RoboDK station: kr30 cnc 072119 not table destroyer.rdk

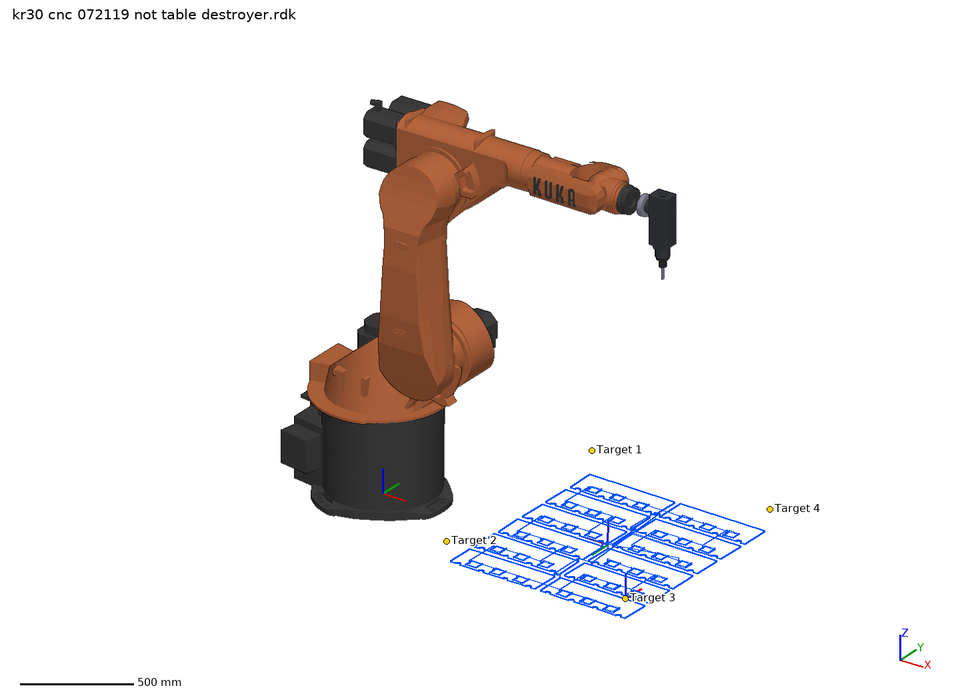
[picture v0: the station drawn from its stored meshes, robots at their saved joint values, targets as dots, program paths as lines]
Station kr30 cnc 072119 not table destroyer. Poses are relative to the parent item; angles as X-Y-Z fixed-axis rotations.
  - frame GIGASHEEN Base at (0, 0, 0) mm
    - robot GIGASHEEN (model KUKA KR 30 HA): 6 axes, payload 30 kg, reach 2033 mm, repeatability 0.05 mm, weight 665 kg
        modified DH rows (alpha deg, a mm, theta deg, d mm): 0, 0, 0, 815; -90, 350, 0, 0; 0, 850, -90, 0; -90, 145, 0, 820; 90, 0, 0, 0; -90, 0, 180, 170
        joint limits [-185, -135, -120, -350, -119, -350] to [185, 35, 158, 350, 119, 350]; home [0, -90, 90, 0, 0, 0]; saved at [0, -90, 90, 0, 0, 0]
      - tool 1/2" End Mill TCP, TCP at (337.71, -2.2, 160.57) mm, rotated rx 0 ry 90 rz 0 deg, size 415.8 x 102 x 153.6 mm
    - target Target 1 (joint target) at (982.46, 202.21, 406.25) mm, rotated rx -179.95 ry 0.15 rz -89.48 deg; joints [7.49, -59.642, 144.935, 97.969, -90.801, -4.608] of GIGASHEEN
    - target Target 2 (joint target) at (986.83, -921.64, 412.07) mm, rotated rx -179.94 ry 0.15 rz -89.48 deg; joints [51.766, -38.608, 94.384, 136.851, -116.554, -22.567] of GIGASHEEN
    - target Target 3 (joint target) at (1949.02, -919.97, 396.91) mm, rotated rx -179.94 ry 0.14 rz 179.61 deg; joints [29.5, -22.76, 62.288, 41.088, -47.759, -30.404] of GIGASHEEN
    - target Target 4 (joint target) at (1949.02, 190.94, 391.63) mm, rotated rx -179.94 ry 0.14 rz 179.61 deg; joints [-6.898, -35.989, 90.741, -8.88, -55.221, 5.167] of GIGASHEEN
  - machining project Machining Settings: C:/Users/liqui/OneDrive/Desktop/first half pipe jig.apt | rotZ(0) | rotX(0)*rotY(0) | rotZ(0)
  - program Prog2 (4 instructions, listed below)
  - frame Table at (1949.02, -919.97, 396.91) mm, rotated rx 0.87 ry 0.27 rz 90 deg
    - frame Frame 4 at (550, 480, -95) mm, rotated rx 0 ry 0 rz 90 deg
  - program Machining (1954 instructions, listed below)
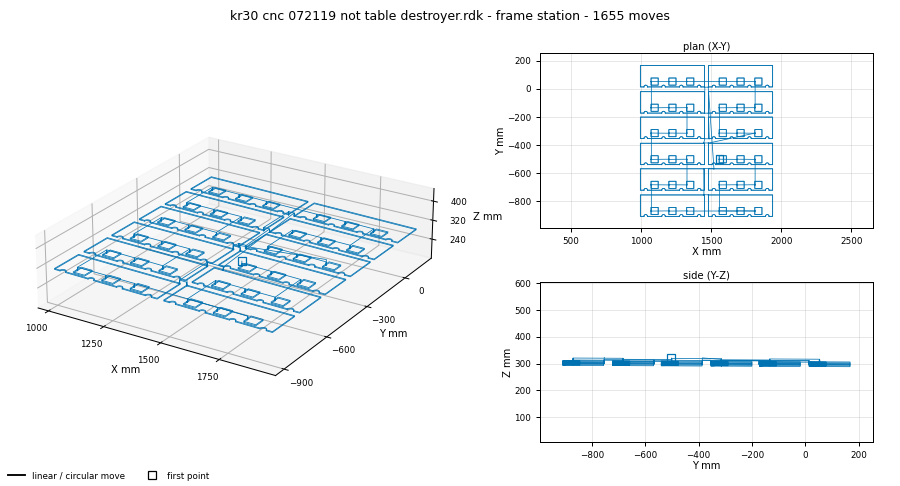
[picture p0: tool path of kr30 cnc 072119 not table destroyer.rdk in frame station, 1655 of 1659 moves have a stored position in this frame; points joined in program order, loops and branches not executed]

--- program Prog2 (robot GIGASHEEN) ---
  MoveJ (plywood back right safe) [its target is no longer in the station]
  MoveL (plywood back left safe) [its target is no longer in the station]
  MoveL (plywood front left safe) [its target is no longer in the station]
  MoveL (plywood front right safe) [its target is no longer in the station]

--- program Machining (robot GIGASHEEN) ---
  Smooth(0)
  Set Ref.: Frame 4
  Set Tool: 1/2" End Mill TCP
  Show 1/2" End Mill TCP
  Print: /'1001'
  Print: /''
  Print: /'2D Contour2'
  Set speed (500.0 mm/s)
  MoveJ 1 to (-92.16, 131.48, 15) mm, rotated rx -180 ry 0 rz 0 deg; joints [21.967, -44.262, 117.716, 22.916, -73.822, -6.095]
  MoveL 2 to (-92.16, 131.48, 15) mm, rotated rx -180 ry 0 rz 0 deg; joints [21.967, -44.262, 117.716, 22.916, -73.822, -6.095]
  MoveL 3 to (-92.16, 131.48, 15) mm, rotated rx -180 ry 0 rz 0 deg; joints [21.967, -44.262, 117.716, 22.916, -73.822, -6.095]
  Set speed (500.0 mm/s)
  MoveL 4 to (-92.16, 131.49, 6) mm, rotated rx -180 ry 0 rz 0 deg; joints [21.971, -43.695, 117.606, 22.87, -74.243, -5.911]
  Set speed (25.4 mm/s)
  MoveL 5 to (-92.16, 131.49, -3.54) mm, rotated rx -180 ry 0 rz 0 deg; joints [21.975, -43.092, 117.482, 22.822, -74.685, -5.719]
  MoveC 6 to (-91.98, 131.48, -3.99) mm, rotated rx -180 ry 0 rz 0 deg; joints [21.978, -43.069, 117.491, 22.822, -74.714, -5.707] to (-91.53, 131.48, -4.17) mm, rotated rx 180 ry 0 rz 0 deg; joints [21.986, -43.07, 117.523, 22.826, -74.743, -5.697]
  Set speed (50.8 mm/s)
  MoveL 7 to (-90.89, 131.48, -4.18) mm, rotated rx -180 ry 0 rz 0 deg; joints [21.996, -43.089, 117.572, 22.834, -74.772, -5.687]
  MoveC 8 to (-90.44, 131.3, -4.18) mm, rotated rx -180 ry 0 rz 0 deg; joints [21.996, -43.104, 117.612, 22.831, -74.796, -5.677] to (-90.26, 130.85, -4.17) mm, rotated rx 180 ry 0 rz 0 deg; joints [21.981, -43.115, 117.641, 22.813, -74.811, -5.666]
  MoveL 9 to (-90.26, 105.45, -4.18) mm, rotated rx -180 ry 0 rz 0 deg; joints [20.958, -43.388, 118.41, 21.71, -75.168, -5.214]
  MoveL 10 to (-141.06, 105.45, -4.18) mm, rotated rx -180 ry 0 rz 0 deg; joints [20.197, -41.862, 114.412, 21.181, -72.789, -5.949]
  MoveL 11 to (-141.06, 156.25, -4.18) mm, rotated rx -180 ry 0 rz 0 deg; joints [22.169, -41.28, 112.846, 23.353, -72.109, -6.929]
  MoveL 12 to (-90.26, 156.25, -4.17) mm, rotated rx -180 ry 0 rz 0 deg; joints [22.989, -42.824, 116.833, 23.909, -74.444, -6.139]
  MoveL 13 to (-90.26, 130.85, -4.17) mm, rotated rx 180 ry 0 rz 0 deg; joints [21.981, -43.115, 117.641, 22.813, -74.811, -5.666]
  MoveC 14 to (-90.44, 130.4, -4.18) mm, rotated rx -180 ry 0 rz 0 deg; joints [21.96, -43.114, 117.64, 22.792, -74.809, -5.661] to (-90.89, 130.21, -4.17) mm, rotated rx 180 ry 0 rz 0 deg; joints [21.945, -43.103, 117.611, 22.779, -74.79, -5.664]
  MoveL 15 to (-91.53, 130.21, -4.18) mm, rotated rx 180 ry 0 rz 0 deg; joints [21.935, -43.085, 117.562, 22.771, -74.761, -5.674]
  MoveC 16 to (-91.98, 130.21, -3.99) mm, rotated rx 180 ry 0 rz 0 deg; joints [21.928, -43.083, 117.53, 22.767, -74.732, -5.684] to (-92.16, 130.21, -3.54) mm, rotated rx -180 ry 0 rz 0 deg; joints [21.925, -43.106, 117.522, 22.767, -74.703, -5.696]
  Set speed (500.0 mm/s)
  MoveL 17 to (-92.16, 130.21, 5) mm, rotated rx 180 ry 0 rz 0 deg; joints [21.921, -43.646, 117.633, 22.809, -74.307, -5.867]
  MoveL 18 to (-92.16, 131.49, 5) mm, rotated rx -180 ry 0 rz 0 deg; joints [21.972, -43.632, 117.594, 22.864, -74.289, -5.891]
  Set speed (25.4 mm/s)
  MoveL 19 to (-92.16, 131.48, 1.82) mm, rotated rx 180 ry 0 rz 0 deg; joints [21.973, -43.431, 117.553, 22.848, -74.437, -5.827]
  MoveL 20 to (-92.16, 131.49, -7.72) mm, rotated rx -180 ry 0 rz 0 deg; joints [21.977, -42.828, 117.425, 22.802, -74.876, -5.636]
  MoveC 21 to (-91.98, 131.48, -8.16) mm, rotated rx -180 ry 0 rz 0 deg; joints [21.98, -42.804, 117.434, 22.802, -74.906, -5.624] to (-91.53, 131.48, -8.35) mm, rotated rx 180 ry 0 rz 0 deg; joints [21.988, -42.806, 117.466, 22.806, -74.935, -5.614]
  Set speed (50.8 mm/s)
  MoveL 22 to (-90.89, 131.48, -8.35) mm, rotated rx -180 ry 0 rz 0 deg; joints [21.998, -42.824, 117.515, 22.814, -74.964, -5.604]
  MoveC 23 to (-90.44, 131.3, -8.35) mm, rotated rx -180 ry 0 rz 0 deg; joints [21.998, -42.839, 117.555, 22.811, -74.988, -5.594] to (-90.26, 130.85, -8.35) mm, rotated rx 180 ry 0 rz 0 deg; joints [21.983, -42.85, 117.584, 22.794, -75.003, -5.583]
  MoveL 24 to (-90.26, 105.45, -8.35) mm, rotated rx -180 ry 0 rz 0 deg; joints [20.96, -43.121, 118.353, 21.691, -75.363, -5.134]
  MoveL 25 to (-141.06, 105.45, -8.35) mm, rotated rx -180 ry 0 rz 0 deg; joints [20.199, -41.606, 114.356, 21.161, -72.976, -5.874]
  MoveL 26 to (-141.06, 156.25, -8.35) mm, rotated rx -180 ry 0 rz 0 deg; joints [22.171, -41.027, 112.79, 23.33, -72.29, -6.848]
  MoveL 27 to (-90.26, 156.25, -8.35) mm, rotated rx -180 ry 0 rz 0 deg; joints [22.991, -42.562, 116.776, 23.888, -74.632, -6.053]
  MoveL 28 to (-90.26, 130.85, -8.35) mm, rotated rx 180 ry 0 rz 0 deg; joints [21.983, -42.85, 117.584, 22.794, -75.003, -5.583]
  MoveC 29 to (-90.44, 130.4, -8.35) mm, rotated rx 180 ry 0 rz 0 deg; joints [21.962, -42.849, 117.583, 22.772, -75.001, -5.578] to (-90.89, 130.21, -8.35) mm, rotated rx -180 ry 0 rz 0 deg; joints [21.947, -42.838, 117.554, 22.759, -74.983, -5.581]
  MoveL 30 to (-91.53, 130.21, -8.35) mm, rotated rx -180 ry 0 rz 0 deg; joints [21.937, -42.82, 117.505, 22.751, -74.953, -5.591]
  MoveC 31 to (-91.98, 130.21, -8.16) mm, rotated rx -180 ry 0 rz 0 deg; joints [21.93, -42.818, 117.473, 22.747, -74.924, -5.601] to (-92.16, 130.21, -7.72) mm, rotated rx 180 ry 0 rz 0 deg; joints [21.926, -42.842, 117.465, 22.747, -74.895, -5.613]
  Set speed (500.0 mm/s)
  MoveL 32 to (-92.16, 130.22, 6) mm, rotated rx -180 ry 0 rz 0 deg; joints [21.92, -43.71, 117.646, 22.814, -74.261, -5.888]
  MoveL 33 to (-219.16, 131.48, 6) mm, rotated rx 180 ry 0 rz 0 deg; joints [20.093, -39.587, 107.343, 21.691, -68.314, -7.771]
  Set speed (25.4 mm/s)
  MoveL 34 to (-219.16, 131.48, -3.54) mm, rotated rx -180 ry 0 rz 0 deg; joints [20.097, -39.042, 107.223, 21.633, -68.71, -7.604]
  MoveC 35 to (-218.98, 131.48, -3.99) mm, rotated rx 180 ry 0 rz 0 deg; joints [20.1, -39.022, 107.233, 21.632, -68.737, -7.593] to (-218.53, 131.48, -4.17) mm, rotated rx -180 ry 0 rz 0 deg; joints [20.106, -39.027, 107.269, 21.634, -68.767, -7.584]
  Set speed (50.8 mm/s)
  MoveL 36 to (-217.89, 131.48, -4.18) mm, rotated rx 180 ry 0 rz 0 deg; joints [20.115, -39.049, 107.322, 21.639, -68.797, -7.574]
  MoveC 37 to (-217.44, 131.3, -4.17) mm, rotated rx -180 ry 0 rz 0 deg; joints [20.114, -39.067, 107.366, 21.634, -68.821, -7.564] to (-217.26, 130.85, -4.17) mm, rotated rx -180 ry 0 rz 0 deg; joints [20.1, -39.079, 107.395, 21.617, -68.836, -7.551]
  MoveL 38 to (-217.26, 105.45, -4.18) mm, rotated rx -180 ry 0 rz 0 deg; joints [19.15, -39.375, 108.156, 20.544, -69.144, -7.025]
  MoveL 39 to (-268.06, 105.45, -4.18) mm, rotated rx 180 ry 0 rz 0 deg; joints [18.508, -37.578, 103.789, 20.221, -66.649, -7.743]
  MoveL 40 to (-268.06, 156.25, -4.18) mm, rotated rx 180 ry 0 rz 0 deg; joints [20.343, -36.949, 102.223, 22.351, -66.05, -8.881]
  MoveL 41 to (-217.26, 156.25, -4.17) mm, rotated rx -180 ry 0 rz 0 deg; joints [21.038, -38.765, 106.595, 22.685, -68.517, -8.097]
  MoveL 42 to (-217.26, 130.85, -4.17) mm, rotated rx -180 ry 0 rz 0 deg; joints [20.1, -39.079, 107.395, 21.617, -68.836, -7.551]
  MoveC 43 to (-217.44, 130.4, -4.17) mm, rotated rx -180 ry 0 rz 0 deg; joints [20.08, -39.078, 107.394, 21.596, -68.832, -7.545] to (-217.89, 130.21, -4.17) mm, rotated rx 180 ry 0 rz 0 deg; joints [20.067, -39.064, 107.361, 21.585, -68.813, -7.547]
  MoveL 44 to (-218.53, 130.21, -4.18) mm, rotated rx -180 ry 0 rz 0 deg; joints [20.059, -39.042, 107.308, 21.581, -68.782, -7.557]
  MoveC 45 to (-218.98, 130.21, -3.99) mm, rotated rx -180 ry 0 rz 0 deg; joints [20.053, -39.038, 107.272, 21.578, -68.753, -7.567] to (-219.16, 130.21, -3.54) mm, rotated rx 180 ry 0 rz 0 deg; joints [20.05, -39.057, 107.262, 21.58, -68.725, -7.577]
  Set speed (500.0 mm/s)
  MoveL 46 to (-219.16, 130.21, 5) mm, rotated rx 180 ry 0 rz 0 deg; joints [20.047, -39.545, 107.37, 21.631, -68.371, -7.727]
  MoveL 47 to (-219.16, 131.48, 5) mm, rotated rx 180 ry 0 rz 0 deg; joints [20.094, -39.53, 107.331, 21.685, -68.355, -7.754]
  Set speed (25.4 mm/s)
  MoveL 48 to (-219.16, 131.48, 1.83) mm, rotated rx -180 ry 0 rz 0 deg; joints [20.095, -39.348, 107.291, 21.666, -68.488, -7.698]
  MoveL 49 to (-219.16, 131.48, -7.72) mm, rotated rx 180 ry 0 rz 0 deg; joints [20.099, -38.802, 107.169, 21.609, -68.882, -7.532]
  MoveC 50 to (-218.98, 131.49, -8.16) mm, rotated rx -180 ry 0 rz 0 deg; joints [20.101, -38.783, 107.179, 21.607, -68.909, -7.521] to (-218.53, 131.48, -8.35) mm, rotated rx -180 ry 0 rz 0 deg; joints [20.108, -38.788, 107.214, 21.609, -68.939, -7.511]
  Set speed (50.8 mm/s)
  MoveL 51 to (-217.89, 131.48, -8.35) mm, rotated rx -180 ry 0 rz 0 deg; joints [20.116, -38.81, 107.268, 21.614, -68.969, -7.502]
  MoveC 52 to (-217.44, 131.3, -8.35) mm, rotated rx 180 ry 0 rz 0 deg; joints [20.115, -38.827, 107.311, 21.61, -68.993, -7.491] to (-217.26, 130.85, -8.35) mm, rotated rx 180 ry 0 rz 0 deg; joints [20.101, -38.839, 107.341, 21.592, -69.008, -7.479]
  MoveL 53 to (-217.26, 105.45, -8.35) mm, rotated rx -180 ry 0 rz 0 deg; joints [19.151, -39.133, 108.101, 20.521, -69.319, -6.956]
  MoveL 54 to (-268.06, 105.45, -8.35) mm, rotated rx -180 ry 0 rz 0 deg; joints [18.509, -37.346, 103.734, 20.196, -66.816, -7.677]
  MoveL 55 to (-268.06, 156.25, -8.35) mm, rotated rx 180 ry 0 rz 0 deg; joints [20.345, -36.72, 102.169, 22.323, -66.212, -8.809]
  MoveL 56 to (-217.26, 156.25, -8.35) mm, rotated rx -180 ry 0 rz 0 deg; joints [21.04, -38.527, 106.541, 22.659, -68.687, -8.021]
  MoveL 57 to (-217.26, 130.85, -8.35) mm, rotated rx 180 ry 0 rz 0 deg; joints [20.101, -38.839, 107.341, 21.592, -69.008, -7.479]
  MoveC 58 to (-217.44, 130.4, -8.35) mm, rotated rx 180 ry 0 rz 0 deg; joints [20.082, -38.838, 107.339, 21.572, -69.005, -7.472] to (-217.89, 130.22, -8.35) mm, rotated rx -180 ry 0 rz 0 deg; joints [20.069, -38.825, 107.307, 21.561, -68.985, -7.475]
  MoveL 59 to (-218.53, 130.22, -8.35) mm, rotated rx -180 ry 0 rz 0 deg; joints [20.06, -38.803, 107.253, 21.556, -68.954, -7.485]
  MoveC 60 to (-218.98, 130.21, -8.16) mm, rotated rx -180 ry 0 rz 0 deg; joints [20.054, -38.798, 107.218, 21.554, -68.925, -7.494] to (-219.16, 130.22, -7.72) mm, rotated rx -180 ry 0 rz 0 deg; joints [20.051, -38.818, 107.208, 21.555, -68.898, -7.505]
  Set speed (500.0 mm/s)
  MoveL 61 to (-219.16, 130.21, 6) mm, rotated rx -180 ry 0 rz 0 deg; joints [20.046, -39.602, 107.382, 21.638, -68.329, -7.744]
  MoveL 62 to (-346.16, 131.48, 6) mm, rotated rx -180 ry 0 rz 0 deg; joints [18.501, -34.783, 96.043, 21.052, -62.014, -9.675]
  Set speed (25.4 mm/s)
  MoveL 63 to (-346.16, 131.48, -3.54) mm, rotated rx -180 ry 0 rz 0 deg; joints [18.504, -34.284, 95.924, 20.984, -62.369, -9.523]
  MoveC 64 to (-345.98, 131.48, -3.99) mm, rotated rx -180 ry 0 rz 0 deg; joints [18.507, -34.269, 95.936, 20.982, -62.395, -9.513] to (-345.53, 131.48, -4.17) mm, rotated rx 180 ry 0 rz 0 deg; joints [18.512, -34.277, 95.975, 20.982, -62.426, -9.503]
  Set speed (50.8 mm/s)
  MoveL 65 to (-344.89, 131.48, -4.18) mm, rotated rx -180 ry 0 rz 0 deg; joints [18.519, -34.303, 96.035, 20.983, -62.458, -9.493]
  MoveC 66 to (-344.44, 131.3, -4.17) mm, rotated rx -180 ry 0 rz 0 deg; joints [18.518, -34.323, 96.083, 20.977, -62.484, -9.481] to (-344.26, 130.85, -4.17) mm, rotated rx -180 ry 0 rz 0 deg; joints [18.504, -34.337, 96.115, 20.959, -62.498, -9.467]
  MoveL 67 to (-344.26, 105.45, -4.18) mm, rotated rx -180 ry 0 rz 0 deg; joints [17.62, -34.658, 96.888, 19.894, -62.777, -8.851]
  MoveL 68 to (-395.06, 105.45, -4.17) mm, rotated rx -180 ry 0 rz 0 deg; joints [17.072, -32.543, 92.01, 19.79, -60.088, -9.633]
  MoveL 69 to (-395.06, 156.25, -4.18) mm, rotated rx -180 ry 0 rz 0 deg; joints [18.786, -31.855, 90.392, 21.931, -59.533, -10.971]
  MoveL 70 to (-344.26, 156.25, -4.18) mm, rotated rx -180 ry 0 rz 0 deg; joints [19.38, -33.996, 95.299, 22.023, -62.209, -10.102]
  MoveL 71 to (-344.26, 130.85, -4.17) mm, rotated rx -180 ry 0 rz 0 deg; joints [18.504, -34.337, 96.115, 20.959, -62.498, -9.467]
  MoveC 72 to (-344.44, 130.4, -4.18) mm, rotated rx -180 ry 0 rz 0 deg; joints [18.487, -34.335, 96.111, 20.939, -62.494, -9.459] to (-344.89, 130.21, -4.18) mm, rotated rx 180 ry 0 rz 0 deg; joints [18.475, -34.319, 96.075, 20.93, -62.473, -9.462]
  MoveL 73 to (-345.53, 130.21, -4.18) mm, rotated rx -180 ry 0 rz 0 deg; joints [18.468, -34.294, 96.015, 20.928, -62.44, -9.472]
  MoveC 74 to (-345.98, 130.22, -3.99) mm, rotated rx -180 ry 0 rz 0 deg; joints [18.463, -34.285, 95.975, 20.928, -62.41, -9.482] to (-346.16, 130.21, -3.54) mm, rotated rx -180 ry 0 rz 0 deg; joints [18.46, -34.301, 95.964, 20.931, -62.383, -9.492]
  Set speed (500.0 mm/s)
  MoveL 75 to (-346.16, 130.21, 5) mm, rotated rx -180 ry 0 rz 0 deg; joints [18.457, -34.748, 96.07, 20.992, -62.065, -9.628]
  MoveL 76 to (-346.16, 131.48, 5) mm, rotated rx -180 ry 0 rz 0 deg; joints [18.501, -34.731, 96.031, 21.045, -62.051, -9.659]
  Set speed (25.4 mm/s)
  MoveL 77 to (-346.16, 131.48, 1.82) mm, rotated rx -180 ry 0 rz 0 deg; joints [18.502, -34.565, 95.992, 21.022, -62.17, -9.608]
  MoveL 78 to (-346.16, 131.48, -7.71) mm, rotated rx 180 ry 0 rz 0 deg; joints [18.506, -34.065, 95.87, 20.955, -62.523, -9.457]
  MoveC 79 to (-345.98, 131.48, -8.16) mm, rotated rx -180 ry 0 rz 0 deg; joints [18.508, -34.049, 95.881, 20.952, -62.549, -9.447] to (-345.53, 131.48, -8.35) mm, rotated rx -180 ry 0 rz 0 deg; joints [18.513, -34.058, 95.921, 20.952, -62.58, -9.437]
  Set speed (50.8 mm/s)
  MoveL 80 to (-344.89, 131.48, -8.35) mm, rotated rx -180 ry 0 rz 0 deg; joints [18.521, -34.083, 95.981, 20.954, -62.613, -9.427]
  MoveC 81 to (-344.44, 131.3, -8.35) mm, rotated rx -180 ry 0 rz 0 deg; joints [18.519, -34.104, 96.029, 20.948, -62.638, -9.415] to (-344.26, 130.85, -8.35) mm, rotated rx 180 ry 0 rz 0 deg; joints [18.506, -34.117, 96.06, 20.93, -62.653, -9.401]
  MoveL 82 to (-344.26, 105.45, -8.35) mm, rotated rx -180 ry 0 rz 0 deg; joints [17.621, -34.437, 96.833, 19.867, -62.934, -8.788]
  MoveL 83 to (-395.06, 105.45, -8.35) mm, rotated rx -180 ry 0 rz 0 deg; joints [17.073, -32.329, 91.955, 19.76, -60.238, -9.572]
  MoveL 84 to (-395.06, 156.25, -8.35) mm, rotated rx -180 ry 0 rz 0 deg; joints [18.787, -31.643, 90.337, 21.899, -59.678, -10.904]
  MoveL 85 to (-344.26, 156.25, -8.35) mm, rotated rx -180 ry 0 rz 0 deg; joints [19.382, -33.778, 95.244, 21.993, -62.361, -10.034]
  MoveL 86 to (-344.26, 130.85, -8.35) mm, rotated rx 180 ry 0 rz 0 deg; joints [18.506, -34.117, 96.06, 20.93, -62.653, -9.401]
  MoveC 87 to (-344.44, 130.4, -8.35) mm, rotated rx -180 ry 0 rz 0 deg; joints [18.488, -34.115, 96.057, 20.91, -62.648, -9.393] to (-344.89, 130.21, -8.35) mm, rotated rx -180 ry 0 rz 0 deg; joints [18.477, -34.1, 96.02, 20.901, -62.627, -9.396]
  MoveL 88 to (-345.53, 130.21, -8.35) mm, rotated rx -180 ry 0 rz 0 deg; joints [18.469, -34.074, 95.961, 20.899, -62.594, -9.406]
  MoveC 89 to (-345.98, 130.21, -8.16) mm, rotated rx -180 ry 0 rz 0 deg; joints [18.464, -34.066, 95.921, 20.899, -62.564, -9.416] to (-346.16, 130.21, -7.72) mm, rotated rx 180 ry 0 rz 0 deg; joints [18.462, -34.082, 95.909, 20.902, -62.538, -9.426]
  Set speed (500.0 mm/s)
  MoveL 90 to (-346.16, 130.21, 6) mm, rotated rx 180 ry 0 rz 0 deg; joints [18.457, -34.8, 96.082, 20.999, -62.028, -9.644]
  MoveL 91 to (-346.16, 313.35, 6) mm, rotated rx -180 ry 0 rz 0 deg; joints [24.551, -31.864, 89.216, 28.735, -59.772, -14.762]
  Set speed (25.4 mm/s)
  MoveL 92 to (-346.16, 313.35, -3.54) mm, rotated rx -180 ry 0 rz 0 deg; joints [24.555, -31.387, 89.095, 28.64, -60.086, -14.565]
  MoveC 93 to (-345.98, 313.35, -3.99) mm, rotated rx -180 ry 0 rz 0 deg; joints [24.557, -31.372, 89.107, 28.636, -60.11, -14.552] to (-345.53, 313.35, -4.17) mm, rotated rx 180 ry 0 rz 0 deg; joints [24.564, -31.382, 89.148, 28.634, -60.139, -14.539]
  Set speed (50.8 mm/s)
  MoveL 94 to (-344.89, 313.35, -4.18) mm, rotated rx 180 ry 0 rz 0 deg; joints [24.573, -31.409, 89.21, 28.635, -60.171, -14.525]
  MoveC 95 to (-344.44, 313.17, -4.18) mm, rotated rx 180 ry 0 rz 0 deg; joints [24.574, -31.432, 89.261, 28.628, -60.197, -14.509] to (-344.26, 312.72, -4.18) mm, rotated rx 180 ry 0 rz 0 deg; joints [24.562, -31.448, 89.299, 28.609, -60.213, -14.491]
  MoveL 96 to (-344.26, 287.32, -4.18) mm, rotated rx -180 ry 0 rz 0 deg; joints [23.747, -31.917, 90.391, 27.535, -60.56, -13.718]
  MoveL 97 to (-395.06, 287.32, -4.17) mm, rotated rx -180 ry 0 rz 0 deg; joints [23.046, -29.688, 85.37, 27.512, -57.909, -14.825]
  MoveL 98 to (-395.06, 338.12, -4.18) mm, rotated rx -180 ry 0 rz 0 deg; joints [24.63, -28.683, 83.075, 29.71, -57.21, -16.501]
  MoveL 99 to (-344.26, 338.12, -4.18) mm, rotated rx -180 ry 0 rz 0 deg; joints [25.367, -30.956, 88.159, 29.688, -59.857, -15.291]
  MoveL 100 to (-344.26, 312.72, -4.17) mm, rotated rx -180 ry 0 rz 0 deg; joints [24.562, -31.448, 89.299, 28.609, -60.213, -14.491]
  MoveC 101 to (-344.44, 312.27, -4.18) mm, rotated rx -180 ry 0 rz 0 deg; joints [24.545, -31.449, 89.301, 28.59, -60.209, -14.481] to (-344.89, 312.08, -4.18) mm, rotated rx -180 ry 0 rz 0 deg; joints [24.533, -31.433, 89.265, 28.581, -60.189, -14.485]
  MoveL 102 to (-345.53, 312.08, -4.17) mm, rotated rx -180 ry 0 rz 0 deg; joints [24.524, -31.406, 89.204, 28.581, -60.157, -14.499]
  MoveC 103 to (-345.98, 312.08, -3.99) mm, rotated rx -180 ry 0 rz 0 deg; joints [24.517, -31.396, 89.163, 28.582, -60.128, -14.513] to (-346.16, 312.08, -3.54) mm, rotated rx -180 ry 0 rz 0 deg; joints [24.514, -31.411, 89.151, 28.586, -60.103, -14.526]
  Set speed (500.0 mm/s)
  MoveL 104 to (-346.16, 312.08, 5) mm, rotated rx -180 ry 0 rz 0 deg; joints [24.511, -31.838, 89.259, 28.671, -59.822, -14.701]
  MoveL 105 to (-346.16, 313.35, 5) mm, rotated rx 180 ry 0 rz 0 deg; joints [24.551, -31.814, 89.203, 28.725, -59.805, -14.741]
  Set speed (25.4 mm/s)
  MoveL 106 to (-346.16, 313.35, 1.82) mm, rotated rx 180 ry 0 rz 0 deg; joints [24.553, -31.655, 89.164, 28.693, -59.91, -14.675]
  MoveL 107 to (-346.16, 313.35, -7.72) mm, rotated rx 180 ry 0 rz 0 deg; joints [24.556, -31.177, 89.04, 28.599, -60.222, -14.481]
  MoveC 108 to (-345.98, 313.35, -8.16) mm, rotated rx -180 ry 0 rz 0 deg; joints [24.559, -31.162, 89.052, 28.595, -60.246, -14.468] to (-345.53, 313.35, -8.35) mm, rotated rx -180 ry 0 rz 0 deg; joints [24.566, -31.172, 89.093, 28.594, -60.275, -14.454]
  Set speed (50.8 mm/s)
  MoveL 109 to (-344.89, 313.35, -8.35) mm, rotated rx -180 ry 0 rz 0 deg; joints [24.575, -31.199, 89.154, 28.595, -60.308, -14.44]
  MoveC 110 to (-344.44, 313.17, -8.35) mm, rotated rx 180 ry 0 rz 0 deg; joints [24.575, -31.221, 89.206, 28.587, -60.333, -14.425] to (-344.26, 312.72, -8.35) mm, rotated rx 180 ry 0 rz 0 deg; joints [24.564, -31.238, 89.244, 28.569, -60.349, -14.407]
  MoveL 111 to (-344.26, 287.32, -8.35) mm, rotated rx -180 ry 0 rz 0 deg; joints [23.749, -31.705, 90.335, 27.496, -60.699, -13.636]
  MoveL 112 to (-395.06, 287.32, -8.35) mm, rotated rx -180 ry 0 rz 0 deg; joints [23.047, -29.482, 85.314, 27.471, -58.042, -14.744]
  MoveL 113 to (-395.06, 338.12, -8.35) mm, rotated rx -180 ry 0 rz 0 deg; joints [24.631, -28.479, 83.018, 29.665, -57.338, -16.416]
  MoveL 114 to (-344.26, 338.12, -8.35) mm, rotated rx 180 ry 0 rz 0 deg; joints [25.369, -30.747, 88.104, 29.645, -59.991, -15.204]
  MoveL 115 to (-344.26, 312.72, -8.35) mm, rotated rx 180 ry 0 rz 0 deg; joints [24.564, -31.238, 89.244, 28.569, -60.349, -14.407]
  MoveC 116 to (-344.44, 312.27, -8.35) mm, rotated rx -180 ry 0 rz 0 deg; joints [24.547, -31.238, 89.245, 28.549, -60.346, -14.397] to (-344.89, 312.08, -8.35) mm, rotated rx -180 ry 0 rz 0 deg; joints [24.534, -31.223, 89.21, 28.541, -60.326, -14.401]
  MoveL 117 to (-345.53, 312.08, -8.35) mm, rotated rx -180 ry 0 rz 0 deg; joints [24.525, -31.196, 89.149, 28.54, -60.293, -14.415]
  MoveC 118 to (-345.98, 312.08, -8.16) mm, rotated rx -180 ry 0 rz 0 deg; joints [24.518, -31.186, 89.108, 28.541, -60.264, -14.428] to (-346.16, 312.08, -7.72) mm, rotated rx 180 ry 0 rz 0 deg; joints [24.516, -31.201, 89.096, 28.545, -60.24, -14.441]
  Set speed (500.0 mm/s)
  MoveL 119 to (-346.16, 312.08, 6) mm, rotated rx 180 ry 0 rz 0 deg; joints [24.511, -31.888, 89.271, 28.681, -59.789, -14.722]
  MoveL 120 to (-219.16, 313.35, 6) mm, rotated rx 180 ry 0 rz 0 deg; joints [26.538, -36.893, 100.706, 29.297, -65.896, -12.2]
  Set speed (25.4 mm/s)
  MoveL 121 to (-219.16, 313.35, -3.54) mm, rotated rx 180 ry 0 rz 0 deg; joints [26.542, -36.378, 100.588, 29.215, -66.244, -11.989]
  MoveC 122 to (-218.98, 313.36, -3.99) mm, rotated rx -180 ry 0 rz 0 deg; joints [26.545, -36.36, 100.598, 29.213, -66.268, -11.976] to (-218.53, 313.36, -4.17) mm, rotated rx -180 ry 0 rz 0 deg; joints [26.553, -36.366, 100.634, 29.214, -66.296, -11.963]
  Set speed (50.8 mm/s)
  MoveL 123 to (-217.89, 313.36, -4.17) mm, rotated rx -180 ry 0 rz 0 deg; joints [26.563, -36.389, 100.688, 29.219, -66.325, -11.951]
  MoveC 124 to (-217.44, 313.17, -4.17) mm, rotated rx -180 ry 0 rz 0 deg; joints [26.565, -36.408, 100.734, 29.215, -66.349, -11.937] to (-217.26, 312.72, -4.17) mm, rotated rx 180 ry 0 rz 0 deg; joints [26.553, -36.423, 100.769, 29.198, -66.364, -11.922]
  MoveL 125 to (-217.26, 287.32, -4.18) mm, rotated rx -180 ry 0 rz 0 deg; joints [25.689, -36.853, 101.821, 28.148, -66.733, -11.243]
  MoveL 126 to (-268.06, 287.32, -4.18) mm, rotated rx 180 ry 0 rz 0 deg; joints [24.878, -34.977, 97.416, 27.815, -64.331, -12.197]
  MoveL 127 to (-268.06, 338.12, -4.18) mm, rotated rx 180 ry 0 rz 0 deg; joints [26.553, -34.068, 95.246, 29.928, -63.609, -13.647]
  MoveL 128 to (-217.26, 338.12, -4.18) mm, rotated rx 180 ry 0 rz 0 deg; joints [27.403, -35.973, 99.674, 30.246, -65.989, -12.625]
  MoveL 129 to (-217.26, 312.72, -4.17) mm, rotated rx 180 ry 0 rz 0 deg; joints [26.553, -36.423, 100.769, 29.198, -66.364, -11.922]
  MoveC 130 to (-217.44, 312.27, -4.17) mm, rotated rx -180 ry 0 rz 0 deg; joints [26.534, -36.424, 100.772, 29.178, -66.362, -11.913] to (-217.89, 312.08, -4.18) mm, rotated rx 180 ry 0 rz 0 deg; joints [26.52, -36.411, 100.742, 29.167, -66.344, -11.917]
  MoveL 131 to (-218.53, 312.08, -4.17) mm, rotated rx -180 ry 0 rz 0 deg; joints [26.51, -36.388, 100.688, 29.162, -66.315, -11.929]
  MoveC 132 to (-218.98, 312.08, -3.99) mm, rotated rx -180 ry 0 rz 0 deg; joints [26.502, -36.382, 100.652, 29.16, -66.287, -11.941] to (-219.16, 312.08, -3.54) mm, rotated rx -180 ry 0 rz 0 deg; joints [26.499, -36.4, 100.642, 29.163, -66.262, -11.955]
  Set speed (500.0 mm/s)
  MoveL 133 to (-219.16, 312.08, 5) mm, rotated rx -180 ry 0 rz 0 deg; joints [26.495, -36.862, 100.748, 29.236, -65.951, -12.143]
  MoveL 134 to (-219.16, 313.35, 5) mm, rotated rx -180 ry 0 rz 0 deg; joints [26.538, -36.839, 100.694, 29.288, -65.932, -12.178]
  Set speed (25.4 mm/s)
  MoveL 135 to (-219.16, 313.35, 1.83) mm, rotated rx -180 ry 0 rz 0 deg; joints [26.539, -36.668, 100.655, 29.261, -66.048, -12.107]
  MoveL 136 to (-219.16, 313.35, -7.71) mm, rotated rx -180 ry 0 rz 0 deg; joints [26.543, -36.151, 100.534, 29.18, -66.395, -11.898]
  MoveC 137 to (-218.98, 313.35, -8.16) mm, rotated rx -180 ry 0 rz 0 deg; joints [26.547, -36.133, 100.544, 29.178, -66.419, -11.885] to (-218.53, 313.35, -8.35) mm, rotated rx -180 ry 0 rz 0 deg; joints [26.554, -36.139, 100.58, 29.179, -66.447, -11.872]
  Set speed (50.8 mm/s)
  MoveL 138 to (-217.89, 313.35, -8.35) mm, rotated rx -180 ry 0 rz 0 deg; joints [26.565, -36.162, 100.634, 29.184, -66.476, -11.86]
  MoveC 139 to (-217.44, 313.17, -8.35) mm, rotated rx -180 ry 0 rz 0 deg; joints [26.566, -36.181, 100.68, 29.18, -66.5, -11.846] to (-217.26, 312.72, -8.35) mm, rotated rx -180 ry 0 rz 0 deg; joints [26.554, -36.196, 100.714, 29.163, -66.515, -11.83]
  MoveL 140 to (-217.26, 287.32, -8.35) mm, rotated rx -180 ry 0 rz 0 deg; joints [25.691, -36.624, 101.767, 28.114, -66.887, -11.154]
  MoveL 141 to (-268.06, 287.32, -8.35) mm, rotated rx -180 ry 0 rz 0 deg; joints [24.88, -34.755, 97.362, 27.78, -64.479, -12.112]
  MoveL 142 to (-268.06, 338.12, -8.35) mm, rotated rx 180 ry 0 rz 0 deg; joints [26.555, -33.85, 95.192, 29.889, -63.751, -13.556]
  MoveL 143 to (-217.26, 338.12, -8.35) mm, rotated rx 180 ry 0 rz 0 deg; joints [27.404, -35.748, 99.62, 30.21, -66.137, -12.531]
  MoveL 144 to (-217.26, 312.72, -8.35) mm, rotated rx -180 ry 0 rz 0 deg; joints [26.554, -36.196, 100.714, 29.163, -66.515, -11.83]
  MoveC 145 to (-217.44, 312.27, -8.35) mm, rotated rx 180 ry 0 rz 0 deg; joints [26.536, -36.197, 100.718, 29.143, -66.513, -11.822] to (-217.89, 312.09, -8.35) mm, rotated rx -180 ry 0 rz 0 deg; joints [26.522, -36.184, 100.687, 29.132, -66.495, -11.825]
  MoveL 146 to (-218.53, 312.08, -8.35) mm, rotated rx 180 ry 0 rz 0 deg; joints [26.511, -36.161, 100.633, 29.127, -66.466, -11.838]
  MoveC 147 to (-218.98, 312.08, -8.16) mm, rotated rx -180 ry 0 rz 0 deg; joints [26.504, -36.155, 100.598, 29.125, -66.438, -11.85] to (-219.16, 312.08, -7.72) mm, rotated rx 180 ry 0 rz 0 deg; joints [26.501, -36.173, 100.588, 29.128, -66.413, -11.864]
  Set speed (500.0 mm/s)
  MoveL 148 to (-219.16, 312.08, 6) mm, rotated rx -180 ry 0 rz 0 deg; joints [26.495, -36.916, 100.76, 29.244, -65.914, -12.165]
  MoveL 149 to (-92.16, 313.35, 6) mm, rotated rx -180 ry 0 rz 0 deg; joints [28.844, -41.18, 110.953, 30.568, -71.515, -9.856]
  Set speed (25.4 mm/s)
  MoveL 150 to (-92.16, 313.35, -3.54) mm, rotated rx -180 ry 0 rz 0 deg; joints [28.849, -40.617, 110.833, 30.498, -71.897, -9.62]
  MoveC 151 to (-91.98, 313.36, -3.99) mm, rotated rx 180 ry 0 rz 0 deg; joints [28.853, -40.596, 110.842, 30.497, -71.923, -9.605] to (-91.53, 313.36, -4.17) mm, rotated rx -180 ry 0 rz 0 deg; joints [28.862, -40.599, 110.874, 30.501, -71.95, -9.593]
  Set speed (50.8 mm/s)
  MoveL 152 to (-90.89, 313.36, -4.18) mm, rotated rx -180 ry 0 rz 0 deg; joints [28.874, -40.618, 110.922, 30.509, -71.977, -9.581]
  MoveC 153 to (-90.44, 313.17, -4.18) mm, rotated rx 180 ry 0 rz 0 deg; joints [28.876, -40.635, 110.964, 30.507, -71.999, -9.568] to (-90.26, 312.72, -4.17) mm, rotated rx 180 ry 0 rz 0 deg; joints [28.864, -40.648, 110.997, 30.491, -72.015, -9.553]
  MoveL 154 to (-90.26, 287.32, -4.18) mm, rotated rx -180 ry 0 rz 0 deg; joints [27.95, -41.048, 112.045, 29.442, -72.424, -8.939]
  MoveL 155 to (-141.06, 287.32, -4.17) mm, rotated rx -180 ry 0 rz 0 deg; joints [27.003, -39.45, 108.078, 28.846, -70.196, -9.855]
  MoveL 156 to (-141.06, 338.12, -4.18) mm, rotated rx 180 ry 0 rz 0 deg; joints [28.775, -38.608, 105.945, 30.937, -69.409, -11.154]
  MoveL 157 to (-90.26, 338.12, -4.17) mm, rotated rx -180 ry 0 rz 0 deg; joints [29.762, -40.229, 109.911, 31.535, -71.6, -10.192]
  MoveL 158 to (-90.26, 312.72, -4.17) mm, rotated rx 180 ry 0 rz 0 deg; joints [28.864, -40.648, 110.997, 30.491, -72.015, -9.553]
  MoveC 159 to (-90.44, 312.27, -4.17) mm, rotated rx -180 ry 0 rz 0 deg; joints [28.844, -40.65, 111.002, 30.47, -72.014, -9.546] to (-90.89, 312.08, -4.18) mm, rotated rx 180 ry 0 rz 0 deg; joints [28.829, -40.639, 110.976, 30.457, -71.998, -9.549]
  MoveL 160 to (-91.53, 312.08, -4.18) mm, rotated rx -180 ry 0 rz 0 deg; joints [28.816, -40.619, 110.927, 30.449, -71.97, -9.561]
  MoveC 161 to (-91.98, 312.08, -3.99) mm, rotated rx 180 ry 0 rz 0 deg; joints [28.808, -40.616, 110.895, 30.445, -71.944, -9.574] to (-92.16, 312.08, -3.54) mm, rotated rx -180 ry 0 rz 0 deg; joints [28.804, -40.637, 110.886, 30.445, -71.918, -9.588]
  Set speed (500.0 mm/s)
  MoveL 162 to (-92.16, 312.08, 5) mm, rotated rx 180 ry 0 rz 0 deg; joints [28.8, -41.142, 110.994, 30.508, -71.575, -9.799]
  MoveL 163 to (-92.16, 313.35, 5) mm, rotated rx -180 ry 0 rz 0 deg; joints [28.845, -41.121, 110.941, 30.56, -71.555, -9.831]
  Set speed (25.4 mm/s)
  MoveL 164 to (-92.16, 313.36, 1.82) mm, rotated rx -180 ry 0 rz 0 deg; joints [28.846, -40.934, 110.902, 30.537, -71.683, -9.752]
  MoveL 165 to (-92.16, 313.35, -7.72) mm, rotated rx -180 ry 0 rz 0 deg; joints [28.851, -40.37, 110.778, 30.468, -72.063, -9.518]
  MoveC 166 to (-91.98, 313.35, -8.16) mm, rotated rx -180 ry 0 rz 0 deg; joints [28.855, -40.349, 110.786, 30.467, -72.089, -9.503] to (-91.53, 313.35, -8.35) mm, rotated rx 180 ry 0 rz 0 deg; joints [28.864, -40.351, 110.818, 30.472, -72.116, -9.491]
  Set speed (50.8 mm/s)
  MoveL 167 to (-90.89, 313.35, -8.35) mm, rotated rx -180 ry 0 rz 0 deg; joints [28.876, -40.371, 110.867, 30.48, -72.143, -9.479]
  MoveC 168 to (-90.44, 313.17, -8.35) mm, rotated rx -180 ry 0 rz 0 deg; joints [28.878, -40.387, 110.909, 30.478, -72.166, -9.466] to (-90.26, 312.72, -8.35) mm, rotated rx -180 ry 0 rz 0 deg; joints [28.866, -40.4, 110.942, 30.462, -72.181, -9.451]
  MoveL 169 to (-90.26, 287.32, -8.35) mm, rotated rx -180 ry 0 rz 0 deg; joints [27.952, -40.798, 111.99, 29.413, -72.594, -8.839]
  MoveL 170 to (-141.06, 287.32, -8.35) mm, rotated rx -180 ry 0 rz 0 deg; joints [27.005, -39.209, 108.023, 28.816, -70.36, -9.76]
  MoveL 171 to (-141.06, 338.12, -8.35) mm, rotated rx -180 ry 0 rz 0 deg; joints [28.777, -38.371, 105.891, 30.904, -69.565, -11.054]
  MoveL 172 to (-90.26, 338.12, -8.35) mm, rotated rx -180 ry 0 rz 0 deg; joints [29.764, -39.984, 109.856, 31.504, -71.763, -10.088]
  MoveL 173 to (-90.26, 312.72, -8.35) mm, rotated rx -180 ry 0 rz 0 deg; joints [28.866, -40.4, 110.942, 30.462, -72.181, -9.451]
  MoveC 174 to (-90.44, 312.27, -8.35) mm, rotated rx -180 ry 0 rz 0 deg; joints [28.846, -40.402, 110.947, 30.441, -72.18, -9.444] to (-90.89, 312.08, -8.35) mm, rotated rx 180 ry 0 rz 0 deg; joints [28.831, -40.391, 110.92, 30.428, -72.164, -9.448]
  MoveL 175 to (-91.53, 312.08, -8.35) mm, rotated rx -180 ry 0 rz 0 deg; joints [28.818, -40.372, 110.872, 30.419, -72.137, -9.459]
  MoveC 176 to (-91.98, 312.08, -8.16) mm, rotated rx -180 ry 0 rz 0 deg; joints [28.809, -40.369, 110.84, 30.415, -72.11, -9.472] to (-92.16, 312.09, -7.72) mm, rotated rx -180 ry 0 rz 0 deg; joints [28.806, -40.39, 110.832, 30.416, -72.084, -9.487]
  Set speed (500.0 mm/s)
  MoveL 177 to (-92.16, 312.08, 6) mm, rotated rx -180 ry 0 rz 0 deg; joints [28.799, -41.201, 111.007, 30.515, -71.535, -9.824]
  MoveL 178 to (-92.16, 499.69, 6) mm, rotated rx 180 ry 0 rz 0 deg; joints [35.058, -37.589, 102.036, 38.119, -68.484, -15.172]
  Set speed (25.4 mm/s)
  MoveL 179 to (-92.16, 499.69, -3.54) mm, rotated rx -180 ry 0 rz 0 deg; joints [35.062, -37.068, 101.919, 38.026, -68.803, -14.906]
  MoveC 180 to (-91.98, 499.69, -3.99) mm, rotated rx 180 ry 0 rz 0 deg; joints [35.067, -37.05, 101.927, 38.024, -68.825, -14.89] to (-91.53, 499.69, -4.17) mm, rotated rx -180 ry 0 rz 0 deg; joints [35.077, -37.054, 101.959, 38.028, -68.85, -14.875]
  Set speed (50.8 mm/s)
  MoveL 181 to (-90.89, 499.69, -4.18) mm, rotated rx -180 ry 0 rz 0 deg; joints [35.09, -37.075, 102.008, 38.035, -68.876, -14.862]
  MoveC 182 to (-90.44, 499.51, -4.18) mm, rotated rx -180 ry 0 rz 0 deg; joints [35.094, -37.094, 102.053, 38.033, -68.897, -14.846] to (-90.26, 499.06, -4.18) mm, rotated rx 180 ry 0 rz 0 deg; joints [35.085, -37.11, 102.091, 38.018, -68.912, -14.828]
  MoveL 183 to (-90.26, 473.66, -4.17) mm, rotated rx 180 ry 0 rz 0 deg; joints [34.286, -37.657, 103.435, 37.006, -69.341, -14.026]
  MoveL 184 to (-141.06, 473.66, -4.18) mm, rotated rx 180 ry 0 rz 0 deg; joints [33.217, -35.965, 99.447, 36.441, -67.227, -15.109]
  MoveL 185 to (-141.06, 524.46, -4.18) mm, rotated rx -180 ry 0 rz 0 deg; joints [34.776, -34.816, 96.694, 38.488, -66.389, -16.788]
  MoveL 186 to (-90.26, 524.46, -4.18) mm, rotated rx -180 ry 0 rz 0 deg; joints [35.868, -36.54, 100.704, 39.026, -68.482, -15.656]
  MoveL 187 to (-90.26, 499.06, -4.18) mm, rotated rx 180 ry 0 rz 0 deg; joints [35.085, -37.11, 102.091, 38.018, -68.912, -14.828]
  MoveC 188 to (-90.44, 498.61, -4.17) mm, rotated rx 180 ry 0 rz 0 deg; joints [35.066, -37.113, 102.101, 37.998, -68.912, -14.817] to (-90.89, 498.42, -4.18) mm, rotated rx 180 ry 0 rz 0 deg; joints [35.051, -37.103, 102.076, 37.985, -68.897, -14.821]
  MoveL 189 to (-91.53, 498.42, -4.18) mm, rotated rx 180 ry 0 rz 0 deg; joints [35.037, -37.082, 102.028, 37.977, -68.871, -14.834]
  MoveC 190 to (-91.98, 498.42, -3.99) mm, rotated rx 180 ry 0 rz 0 deg; joints [35.027, -37.078, 101.995, 37.974, -68.847, -14.849] to (-92.16, 498.42, -3.54) mm, rotated rx 180 ry 0 rz 0 deg; joints [35.023, -37.096, 101.987, 37.976, -68.824, -14.866]
  Set speed (500.0 mm/s)
  MoveL 191 to (-92.16, 498.42, 5) mm, rotated rx 180 ry 0 rz 0 deg; joints [35.019, -37.563, 102.093, 38.058, -68.539, -15.103]
  MoveL 192 to (-92.16, 499.69, 5) mm, rotated rx 180 ry 0 rz 0 deg; joints [35.058, -37.535, 102.024, 38.109, -68.518, -15.144]
  Set speed (25.4 mm/s)
  MoveL 193 to (-92.16, 499.69, 1.82) mm, rotated rx -180 ry 0 rz 0 deg; joints [35.06, -37.362, 101.986, 38.078, -68.624, -15.055]
  MoveL 194 to (-92.16, 499.69, -7.71) mm, rotated rx 180 ry 0 rz 0 deg; joints [35.064, -36.839, 101.865, 37.987, -68.941, -14.792]
  MoveC 195 to (-91.98, 499.69, -8.16) mm, rotated rx 180 ry 0 rz 0 deg; joints [35.069, -36.821, 101.873, 37.985, -68.964, -14.775] to (-91.53, 499.69, -8.35) mm, rotated rx -180 ry 0 rz 0 deg; joints [35.079, -36.825, 101.905, 37.988, -68.988, -14.76]
  Set speed (50.8 mm/s)
  MoveL 196 to (-90.89, 499.69, -8.35) mm, rotated rx -180 ry 0 rz 0 deg; joints [35.092, -36.846, 101.954, 37.996, -69.014, -14.747]
  MoveC 197 to (-90.44, 499.51, -8.35) mm, rotated rx -180 ry 0 rz 0 deg; joints [35.096, -36.864, 101.999, 37.994, -69.036, -14.731] to (-90.26, 499.06, -8.35) mm, rotated rx 180 ry 0 rz 0 deg; joints [35.087, -36.88, 102.037, 37.978, -69.051, -14.713]
  MoveL 198 to (-90.26, 473.66, -8.35) mm, rotated rx 180 ry 0 rz 0 deg; joints [34.288, -37.426, 103.381, 36.968, -69.484, -13.913]
  MoveL 199 to (-141.06, 473.66, -8.35) mm, rotated rx -180 ry 0 rz 0 deg; joints [33.219, -35.741, 99.393, 36.401, -67.365, -15]
  MoveL 200 to (-141.06, 524.46, -8.35) mm, rotated rx -180 ry 0 rz 0 deg; joints [34.778, -34.596, 96.64, 38.445, -66.52, -16.676]
  MoveL 201 to (-90.26, 524.46, -8.35) mm, rotated rx -180 ry 0 rz 0 deg; joints [35.87, -36.313, 100.65, 38.985, -68.617, -15.54]
  MoveL 202 to (-90.26, 499.06, -8.35) mm, rotated rx 180 ry 0 rz 0 deg; joints [35.087, -36.88, 102.037, 37.978, -69.051, -14.713]
  MoveC 203 to (-90.44, 498.61, -8.35) mm, rotated rx 180 ry 0 rz 0 deg; joints [35.068, -36.884, 102.047, 37.958, -69.051, -14.702] to (-90.89, 498.42, -8.35) mm, rotated rx 180 ry 0 rz 0 deg; joints [35.053, -36.874, 102.022, 37.946, -69.036, -14.706]
  MoveL 204 to (-91.53, 498.42, -8.35) mm, rotated rx 180 ry 0 rz 0 deg; joints [35.039, -36.853, 101.974, 37.938, -69.01, -14.72]
  MoveC 205 to (-91.98, 498.42, -8.16) mm, rotated rx -180 ry 0 rz 0 deg; joints [35.029, -36.849, 101.941, 37.934, -68.985, -14.735] to (-92.16, 498.42, -7.72) mm, rotated rx -180 ry 0 rz 0 deg; joints [35.025, -36.867, 101.933, 37.936, -68.963, -14.751]
  Set speed (500.0 mm/s)
  MoveL 206 to (-92.16, 498.42, 6) mm, rotated rx 180 ry 0 rz 0 deg; joints [35.018, -37.617, 102.105, 38.068, -68.505, -15.131]
  MoveL 207 to (-219.16, 499.69, 6) mm, rotated rx -180 ry 0 rz 0 deg; joints [32.467, -33.047, 91.63, 37.007, -63.083, -18.015]
  Set speed (25.4 mm/s)
  MoveL 208 to (-219.16, 499.69, -3.54) mm, rotated rx -180 ry 0 rz 0 deg; joints [32.471, -32.563, 91.511, 36.9, -63.376, -17.771]
  MoveC 209 to (-218.98, 499.69, -3.99) mm, rotated rx -180 ry 0 rz 0 deg; joints [32.475, -32.547, 91.522, 36.896, -63.398, -17.755] to (-218.53, 499.69, -4.17) mm, rotated rx 180 ry 0 rz 0 deg; joints [32.484, -32.555, 91.558, 36.897, -63.424, -17.74]
  Set speed (50.8 mm/s)
  MoveL 210 to (-217.89, 499.69, -4.18) mm, rotated rx -180 ry 0 rz 0 deg; joints [32.496, -32.579, 91.614, 36.9, -63.452, -17.724]
  MoveC 211 to (-217.44, 499.51, -4.17) mm, rotated rx -180 ry 0 rz 0 deg; joints [32.499, -32.601, 91.663, 36.895, -63.476, -17.707] to (-217.26, 499.06, -4.18) mm, rotated rx 180 ry 0 rz 0 deg; joints [32.489, -32.619, 91.705, 36.878, -63.491, -17.687]
  MoveL 212 to (-217.26, 473.66, -4.18) mm, rotated rx -180 ry 0 rz 0 deg; joints [31.721, -33.209, 93.086, 35.829, -63.897, -16.813]
  MoveL 213 to (-268.06, 473.66, -4.18) mm, rotated rx 180 ry 0 rz 0 deg; joints [30.789, -31.208, 88.552, 35.592, -61.557, -18.033]
  MoveL 214 to (-268.06, 524.46, -4.17) mm, rotated rx 180 ry 0 rz 0 deg; joints [32.288, -29.955, 85.676, 37.742, -60.749, -19.897]
  MoveL 215 to (-217.26, 524.46, -4.18) mm, rotated rx 180 ry 0 rz 0 deg; joints [33.244, -32.003, 90.273, 37.929, -63.081, -18.591]
  MoveL 216 to (-217.26, 499.06, -4.18) mm, rotated rx 180 ry 0 rz 0 deg; joints [32.489, -32.619, 91.705, 36.878, -63.491, -17.687]
  MoveC 217 to (-217.44, 498.61, -4.17) mm, rotated rx -180 ry 0 rz 0 deg; joints [32.472, -32.622, 91.713, 36.858, -63.49, -17.676] to (-217.89, 498.42, -4.18) mm, rotated rx -180 ry 0 rz 0 deg; joints [32.458, -32.609, 91.684, 36.848, -63.473, -17.68]
  MoveL 218 to (-218.53, 498.42, -4.18) mm, rotated rx 180 ry 0 rz 0 deg; joints [32.446, -32.585, 91.629, 36.844, -63.444, -17.695]
  MoveC 219 to (-218.98, 498.42, -3.99) mm, rotated rx -180 ry 0 rz 0 deg; joints [32.437, -32.577, 91.592, 36.844, -63.418, -17.711] to (-219.16, 498.42, -3.54) mm, rotated rx -180 ry 0 rz 0 deg; joints [32.433, -32.593, 91.582, 36.848, -63.396, -17.727]
  Set speed (500.0 mm/s)
  MoveL 220 to (-219.16, 498.42, 5) mm, rotated rx 180 ry 0 rz 0 deg; joints [32.43, -33.027, 91.688, 36.943, -63.134, -17.945]
  MoveL 221 to (-219.16, 499.69, 5) mm, rotated rx 180 ry 0 rz 0 deg; joints [32.468, -32.996, 91.618, 36.995, -63.114, -17.989]
  Set speed (25.4 mm/s)
  MoveL 222 to (-219.16, 499.69, 1.82) mm, rotated rx -180 ry 0 rz 0 deg; joints [32.469, -32.835, 91.579, 36.96, -63.211, -17.908]
  MoveL 223 to (-219.16, 499.69, -7.71) mm, rotated rx -180 ry 0 rz 0 deg; joints [32.473, -32.35, 91.457, 36.855, -63.503, -17.666]
  MoveC 224 to (-218.98, 499.69, -8.16) mm, rotated rx 180 ry 0 rz 0 deg; joints [32.477, -32.334, 91.467, 36.851, -63.525, -17.65] to (-218.53, 499.69, -8.35) mm, rotated rx 180 ry 0 rz 0 deg; joints [32.486, -32.342, 91.504, 36.851, -63.551, -17.634]
  Set speed (50.8 mm/s)
  MoveL 225 to (-217.89, 499.69, -8.35) mm, rotated rx -180 ry 0 rz 0 deg; joints [32.498, -32.366, 91.559, 36.855, -63.58, -17.619]
  MoveC 226 to (-217.44, 499.51, -8.35) mm, rotated rx -180 ry 0 rz 0 deg; joints [32.501, -32.388, 91.609, 36.85, -63.603, -17.602] to (-217.26, 499.06, -8.35) mm, rotated rx 180 ry 0 rz 0 deg; joints [32.491, -32.406, 91.65, 36.832, -63.618, -17.582]
  MoveL 227 to (-217.26, 473.66, -8.35) mm, rotated rx -180 ry 0 rz 0 deg; joints [31.723, -32.994, 93.032, 35.785, -64.028, -16.71]
  MoveL 228 to (-268.06, 473.66, -8.35) mm, rotated rx 180 ry 0 rz 0 deg; joints [30.791, -30.999, 88.497, 35.545, -61.683, -17.932]
  MoveL 229 to (-268.06, 524.46, -8.35) mm, rotated rx 180 ry 0 rz 0 deg; joints [32.29, -29.749, 85.62, 37.692, -60.868, -19.792]
  MoveL 230 to (-217.26, 524.46, -8.35) mm, rotated rx -180 ry 0 rz 0 deg; joints [33.246, -31.792, 90.218, 37.882, -63.205, -18.484]
  MoveL 231 to (-217.26, 499.06, -8.35) mm, rotated rx 180 ry 0 rz 0 deg; joints [32.491, -32.406, 91.65, 36.832, -63.618, -17.582]
  MoveC 232 to (-217.44, 498.61, -8.35) mm, rotated rx -180 ry 0 rz 0 deg; joints [32.474, -32.409, 91.659, 36.813, -63.617, -17.57] to (-217.89, 498.42, -8.35) mm, rotated rx 180 ry 0 rz 0 deg; joints [32.46, -32.396, 91.63, 36.802, -63.6, -17.575]
  MoveL 233 to (-218.53, 498.42, -8.35) mm, rotated rx -180 ry 0 rz 0 deg; joints [32.448, -32.372, 91.574, 36.799, -63.572, -17.59]
  MoveC 234 to (-218.98, 498.42, -8.16) mm, rotated rx -180 ry 0 rz 0 deg; joints [32.439, -32.364, 91.537, 36.798, -63.546, -17.605] to (-219.16, 498.42, -7.72) mm, rotated rx -180 ry 0 rz 0 deg; joints [32.435, -32.38, 91.527, 36.802, -63.524, -17.621]
  Set speed (500.0 mm/s)
  MoveL 235 to (-219.16, 498.42, 6) mm, rotated rx -180 ry 0 rz 0 deg; joints [32.429, -33.077, 91.701, 36.954, -63.103, -17.97]
  MoveL 236 to (-346.16, 499.69, 6) mm, rotated rx 180 ry 0 rz 0 deg; joints [30.199, -27.635, 79.633, 36.823, -57.04, -21.385]
  Set speed (25.4 mm/s)
  MoveL 237 to (-346.16, 499.69, -3.54) mm, rotated rx -180 ry 0 rz 0 deg; joints [30.203, -27.18, 79.507, 36.7, -57.305, -21.153]
  MoveC 238 to (-345.98, 499.69, -3.99) mm, rotated rx -180 ry 0 rz 0 deg; joints [30.206, -27.168, 79.52, 36.694, -57.327, -21.137] to (-345.53, 499.69, -4.17) mm, rotated rx -180 ry 0 rz 0 deg; joints [30.214, -27.18, 79.564, 36.691, -57.355, -21.119]
  Set speed (50.8 mm/s)
  MoveL 239 to (-344.89, 499.69, -4.18) mm, rotated rx 180 ry 0 rz 0 deg; joints [30.224, -27.209, 79.629, 36.689, -57.387, -21.1]
  MoveC 240 to (-344.44, 499.51, -4.17) mm, rotated rx 180 ry 0 rz 0 deg; joints [30.226, -27.235, 79.686, 36.679, -57.413, -21.079] to (-344.26, 499.06, -4.17) mm, rotated rx -180 ry 0 rz 0 deg; joints [30.217, -27.256, 79.732, 36.659, -57.43, -21.055]
  MoveL 241 to (-344.26, 473.66, -4.18) mm, rotated rx -180 ry 0 rz 0 deg; joints [29.48, -27.913, 81.211, 35.537, -57.832, -20.057]
  MoveL 242 to (-395.06, 473.66, -4.17) mm, rotated rx -180 ry 0 rz 0 deg; joints [28.663, -25.478, 75.869, 35.743, -55.175, -21.596]
  MoveL 243 to (-395.06, 524.46, -4.18) mm, rotated rx 180 ry 0 rz 0 deg; joints [30.1, -24.05, 72.704, 38.101, -54.347, -23.787]
  MoveL 244 to (-344.26, 524.46, -4.18) mm, rotated rx 180 ry 0 rz 0 deg; joints [30.942, -26.568, 78.19, 37.792, -57.02, -22.092]
  MoveL 245 to (-344.26, 499.06, -4.17) mm, rotated rx -180 ry 0 rz 0 deg; joints [30.217, -27.256, 79.732, 36.659, -57.43, -21.055]
  MoveC 246 to (-344.44, 498.61, -4.17) mm, rotated rx -180 ry 0 rz 0 deg; joints [30.201, -27.259, 79.739, 36.639, -57.427, -21.043] to (-344.89, 498.42, -4.18) mm, rotated rx -180 ry 0 rz 0 deg; joints [30.188, -27.243, 79.704, 36.632, -57.408, -21.049]
  MoveL 247 to (-345.53, 498.42, -4.18) mm, rotated rx 180 ry 0 rz 0 deg; joints [30.177, -27.213, 79.639, 36.634, -57.375, -21.068]
  MoveC 248 to (-345.98, 498.42, -3.99) mm, rotated rx -180 ry 0 rz 0 deg; joints [30.17, -27.201, 79.596, 36.638, -57.347, -21.086] to (-346.16, 498.42, -3.54) mm, rotated rx 180 ry 0 rz 0 deg; joints [30.166, -27.214, 79.583, 36.644, -57.325, -21.102]
  Set speed (500.0 mm/s)
  MoveL 249 to (-346.16, 498.42, 5) mm, rotated rx 180 ry 0 rz 0 deg; joints [30.163, -27.622, 79.696, 36.754, -57.088, -21.309]
  MoveL 250 to (-346.16, 499.69, 5) mm, rotated rx 180 ry 0 rz 0 deg; joints [30.199, -27.588, 79.62, 36.81, -57.068, -21.361]
  Set speed (25.4 mm/s)
  MoveL 251 to (-346.16, 499.69, 1.82) mm, rotated rx 180 ry 0 rz 0 deg; joints [30.201, -27.437, 79.579, 36.769, -57.156, -21.283]
  MoveL 252 to (-346.16, 499.69, -7.72) mm, rotated rx 180 ry 0 rz 0 deg; joints [30.204, -26.98, 79.45, 36.648, -57.42, -21.053]
  MoveC 253 to (-345.98, 499.69, -8.16) mm, rotated rx -180 ry 0 rz 0 deg; joints [30.208, -26.967, 79.462, 36.642, -57.442, -21.037] to (-345.53, 499.69, -8.35) mm, rotated rx -180 ry 0 rz 0 deg; joints [30.215, -26.979, 79.506, 36.638, -57.47, -21.019]
  Set speed (50.8 mm/s)
  MoveL 254 to (-344.89, 499.69, -8.35) mm, rotated rx -180 ry 0 rz 0 deg; joints [30.226, -27.009, 79.571, 36.636, -57.502, -21]
  MoveC 255 to (-344.44, 499.51, -8.35) mm, rotated rx -180 ry 0 rz 0 deg; joints [30.228, -27.035, 79.628, 36.627, -57.528, -20.979] to (-344.26, 499.06, -8.35) mm, rotated rx 180 ry 0 rz 0 deg; joints [30.218, -27.055, 79.674, 36.606, -57.545, -20.955]
  MoveL 256 to (-344.26, 473.66, -8.35) mm, rotated rx -180 ry 0 rz 0 deg; joints [29.482, -27.711, 81.154, 35.486, -57.951, -19.958]
  MoveL 257 to (-395.06, 473.66, -8.35) mm, rotated rx 180 ry 0 rz 0 deg; joints [28.664, -25.281, 75.809, 35.689, -55.287, -21.499]
  MoveL 258 to (-395.06, 524.46, -8.35) mm, rotated rx -180 ry 0 rz 0 deg; joints [30.102, -23.855, 72.643, 38.044, -54.454, -23.686]
  MoveL 259 to (-344.26, 524.46, -8.35) mm, rotated rx -180 ry 0 rz 0 deg; joints [30.944, -26.369, 78.132, 37.738, -57.132, -21.99]
  MoveL 260 to (-344.26, 499.06, -8.35) mm, rotated rx 180 ry 0 rz 0 deg; joints [30.218, -27.055, 79.674, 36.606, -57.545, -20.955]
  MoveC 261 to (-344.44, 498.61, -8.35) mm, rotated rx 180 ry 0 rz 0 deg; joints [30.202, -27.058, 79.682, 36.587, -57.543, -20.943] to (-344.89, 498.42, -8.35) mm, rotated rx 180 ry 0 rz 0 deg; joints [30.189, -27.042, 79.647, 36.58, -57.523, -20.949]
  MoveL 262 to (-345.53, 498.42, -8.35) mm, rotated rx 180 ry 0 rz 0 deg; joints [30.179, -27.013, 79.581, 36.582, -57.49, -20.968]
  MoveC 263 to (-345.98, 498.42, -8.16) mm, rotated rx -180 ry 0 rz 0 deg; joints [30.171, -27.001, 79.538, 36.585, -57.462, -20.986] to (-346.16, 498.42, -7.72) mm, rotated rx -180 ry 0 rz 0 deg; joints [30.168, -27.014, 79.525, 36.591, -57.44, -21.002]
  Set speed (500.0 mm/s)
  MoveL 264 to (-346.16, 498.42, 6) mm, rotated rx -180 ry 0 rz 0 deg; joints [30.163, -27.669, 79.708, 36.767, -57.06, -21.334]
  MoveL 265 to (139.15, 499.69, 6) mm, rotated rx 180 ry 0 rz 0 deg; joints [40.81, -44.208, 118.154, 42.101, -77.062, -10.414]
  Set speed (25.4 mm/s)
  MoveL 266 to (139.15, 499.69, -3.54) mm, rotated rx -180 ry 0 rz 0 deg; joints [40.815, -43.602, 118.031, 42.033, -77.422, -10.083]
  MoveC 267 to (139.34, 499.69, -3.99) mm, rotated rx -180 ry 0 rz 0 deg; joints [40.821, -43.578, 118.036, 42.035, -77.445, -10.064] to (139.79, 499.69, -4.17) mm, rotated rx -180 ry 0 rz 0 deg; joints [40.834, -43.577, 118.062, 42.043, -77.467, -10.048]
  Set speed (50.8 mm/s)
  MoveL 268 to (140.42, 499.69, -4.17) mm, rotated rx -180 ry 0 rz 0 deg; joints [40.852, -43.592, 118.102, 42.058, -77.489, -10.035]
  MoveC 269 to (140.87, 499.51, -4.17) mm, rotated rx -180 ry 0 rz 0 deg; joints [40.858, -43.607, 118.14, 42.061, -77.508, -10.02] to (141.06, 499.06, -4.18) mm, rotated rx 180 ry 0 rz 0 deg; joints [40.849, -43.62, 118.176, 42.048, -77.523, -10.002]
  MoveL 270 to (141.06, 473.66, -4.17) mm, rotated rx -180 ry 0 rz 0 deg; joints [40.007, -44.109, 119.535, 41.074, -78.029, -9.245]
  MoveL 271 to (90.26, 473.66, -4.18) mm, rotated rx -180 ry 0 rz 0 deg; joints [38.617, -42.856, 116.258, 39.971, -76.248, -10.303]
  MoveL 272 to (90.26, 524.46, -4.18) mm, rotated rx -180 ry 0 rz 0 deg; joints [40.267, -41.832, 113.525, 41.924, -75.281, -11.844]
  MoveL 273 to (141.06, 524.46, -4.17) mm, rotated rx 180 ry 0 rz 0 deg; joints [41.67, -43.11, 116.783, 43.011, -77.023, -10.785]
  MoveL 274 to (141.06, 499.06, -4.18) mm, rotated rx 180 ry 0 rz 0 deg; joints [40.849, -43.62, 118.176, 42.048, -77.523, -10.002]
  MoveC 275 to (140.87, 498.61, -4.17) mm, rotated rx 180 ry 0 rz 0 deg; joints [40.829, -43.624, 118.189, 42.027, -77.526, -9.993] to (140.42, 498.42, -4.18) mm, rotated rx -180 ry 0 rz 0 deg; joints [40.81, -43.617, 118.171, 42.009, -77.514, -9.996]
  MoveL 276 to (139.79, 498.42, -4.18) mm, rotated rx -180 ry 0 rz 0 deg; joints [40.792, -43.602, 118.131, 41.995, -77.492, -10.01]
  MoveC 277 to (139.34, 498.42, -3.99) mm, rotated rx -180 ry 0 rz 0 deg; joints [40.779, -43.603, 118.105, 41.986, -77.47, -10.026] to (139.15, 498.42, -3.54) mm, rotated rx 180 ry 0 rz 0 deg; joints [40.774, -43.627, 118.099, 41.985, -77.447, -10.045]
  Set speed (500.0 mm/s)
  MoveL 278 to (139.15, 498.42, 5) mm, rotated rx 180 ry 0 rz 0 deg; joints [40.769, -44.17, 118.21, 42.045, -77.125, -10.341]
  MoveL 279 to (139.15, 499.69, 5) mm, rotated rx -180 ry 0 rz 0 deg; joints [40.81, -44.145, 118.141, 42.094, -77.1, -10.379]
  Set speed (25.4 mm/s)
  MoveL 280 to (139.15, 499.69, 1.82) mm, rotated rx -180 ry 0 rz 0 deg; joints [40.812, -43.943, 118.101, 42.071, -77.22, -10.269]
  MoveL 281 to (139.15, 499.69, -7.71) mm, rotated rx 180 ry 0 rz 0 deg; joints [40.818, -43.336, 117.974, 42.005, -77.578, -9.94]
  MoveC 282 to (139.34, 499.69, -8.16) mm, rotated rx -180 ry 0 rz 0 deg; joints [40.823, -43.312, 117.98, 42.006, -77.601, -9.921] to (139.79, 499.69, -8.35) mm, rotated rx 180 ry 0 rz 0 deg; joints [40.836, -43.311, 118.005, 42.015, -77.623, -9.905]
  Set speed (50.8 mm/s)
  MoveL 283 to (140.42, 499.69, -8.35) mm, rotated rx -180 ry 0 rz 0 deg; joints [40.854, -43.326, 118.045, 42.029, -77.645, -9.892]
  MoveC 284 to (140.87, 499.51, -8.35) mm, rotated rx -180 ry 0 rz 0 deg; joints [40.861, -43.34, 118.084, 42.033, -77.664, -9.877] to (141.06, 499.06, -8.35) mm, rotated rx -180 ry 0 rz 0 deg; joints [40.851, -43.354, 118.12, 42.02, -77.679, -9.859]
  MoveL 285 to (141.06, 473.66, -8.35) mm, rotated rx -180 ry 0 rz 0 deg; joints [40.009, -43.838, 119.477, 41.047, -78.19, -9.102]
  MoveL 286 to (90.26, 473.66, -8.35) mm, rotated rx -180 ry 0 rz 0 deg; joints [38.619, -42.595, 116.202, 39.941, -76.406, -10.168]
  MoveL 287 to (90.26, 524.46, -8.35) mm, rotated rx -180 ry 0 rz 0 deg; joints [40.269, -41.578, 113.469, 41.892, -75.429, -11.708]
  MoveL 288 to (141.06, 524.46, -8.35) mm, rotated rx 180 ry 0 rz 0 deg; joints [41.673, -42.848, 116.726, 42.981, -77.175, -10.641]
  MoveL 289 to (141.06, 499.06, -8.35) mm, rotated rx 180 ry 0 rz 0 deg; joints [40.851, -43.354, 118.12, 42.02, -77.679, -9.859]
  MoveC 290 to (140.87, 498.61, -8.35) mm, rotated rx -180 ry 0 rz 0 deg; joints [40.831, -43.358, 118.132, 41.998, -77.682, -9.849] to (140.42, 498.42, -8.35) mm, rotated rx -180 ry 0 rz 0 deg; joints [40.813, -43.351, 118.114, 41.981, -77.67, -9.853]
  MoveL 291 to (139.79, 498.42, -8.35) mm, rotated rx 180 ry 0 rz 0 deg; joints [40.795, -43.336, 118.074, 41.967, -77.649, -9.867]
  MoveC 292 to (139.34, 498.42, -8.16) mm, rotated rx -180 ry 0 rz 0 deg; joints [40.782, -43.337, 118.048, 41.958, -77.627, -9.882] to (139.15, 498.42, -7.72) mm, rotated rx -180 ry 0 rz 0 deg; joints [40.776, -43.361, 118.043, 41.956, -77.603, -9.902]
  Set speed (500.0 mm/s)
  MoveL 293 to (139.15, 498.42, 6) mm, rotated rx -180 ry 0 rz 0 deg; joints [40.768, -44.234, 118.223, 42.052, -77.087, -10.375]
  MoveL 294 to (266.15, 499.69, 6) mm, rotated rx -180 ry 0 rz 0 deg; joints [44.672, -47.064, 125.748, 45.353, -81.117, -7.753]
  Set speed (25.4 mm/s)
  MoveL 295 to (266.15, 499.69, -3.54) mm, rotated rx -180 ry 0 rz 0 deg; joints [44.678, -46.4, 125.618, 45.301, -81.494, -7.37]
  MoveC 296 to (266.34, 499.69, -3.99) mm, rotated rx -180 ry 0 rz 0 deg; joints [44.684, -46.372, 125.623, 45.304, -81.517, -7.348] to (266.79, 499.69, -4.17) mm, rotated rx 180 ry 0 rz 0 deg; joints [44.699, -46.368, 125.645, 45.316, -81.538, -7.331]
  Set speed (50.8 mm/s)
  MoveL 297 to (267.42, 499.69, -4.17) mm, rotated rx -180 ry 0 rz 0 deg; joints [44.72, -46.381, 125.681, 45.334, -81.557, -7.317]
  MoveC 298 to (267.87, 499.51, -4.17) mm, rotated rx -180 ry 0 rz 0 deg; joints [44.729, -46.393, 125.717, 45.34, -81.574, -7.301] to (268.06, 499.06, -4.17) mm, rotated rx -180 ry 0 rz 0 deg; joints [44.72, -46.405, 125.752, 45.329, -81.59, -7.283]
  MoveL 299 to (268.06, 473.66, -4.18) mm, rotated rx 180 ry 0 rz 0 deg; joints [43.867, -46.858, 127.148, 44.379, -82.151, -6.503]
  MoveL 300 to (217.26, 473.66, -4.17) mm, rotated rx -180 ry 0 rz 0 deg; joints [42.253, -45.823, 124.199, 42.961, -80.561, -7.621]
  MoveL 301 to (217.26, 524.46, -4.18) mm, rotated rx -180 ry 0 rz 0 deg; joints [43.931, -44.866, 121.409, 44.869, -79.493, -9.178]
  MoveL 302 to (268.06, 524.46, -4.17) mm, rotated rx -180 ry 0 rz 0 deg; joints [45.548, -45.93, 124.324, 46.263, -81.04, -8.087]
  MoveL 303 to (268.06, 499.06, -4.17) mm, rotated rx -180 ry 0 rz 0 deg; joints [44.72, -46.405, 125.752, 45.329, -81.59, -7.283]
  MoveC 304 to (267.87, 498.61, -4.18) mm, rotated rx 180 ry 0 rz 0 deg; joints [44.699, -46.41, 125.767, 45.307, -81.594, -7.273] to (267.42, 498.42, -4.18) mm, rotated rx -180 ry 0 rz 0 deg; joints [44.678, -46.404, 125.752, 45.287, -81.584, -7.277]
  MoveL 305 to (266.79, 498.42, -4.18) mm, rotated rx -180 ry 0 rz 0 deg; joints [44.657, -46.392, 125.716, 45.269, -81.565, -7.291]
  MoveC 306 to (266.34, 498.42, -3.99) mm, rotated rx -180 ry 0 rz 0 deg; joints [44.642, -46.396, 125.693, 45.257, -81.545, -7.308] to (266.15, 498.42, -3.54) mm, rotated rx 180 ry 0 rz 0 deg; joints [44.636, -46.423, 125.689, 45.254, -81.521, -7.33]
  Set speed (500.0 mm/s)
  MoveL 307 to (266.15, 498.42, 5) mm, rotated rx -180 ry 0 rz 0 deg; joints [44.63, -47.018, 125.806, 45.3, -81.184, -7.673]
  MoveL 308 to (266.15, 499.69, 5) mm, rotated rx -180 ry 0 rz 0 deg; joints [44.672, -46.994, 125.735, 45.347, -81.157, -7.713]
  Set speed (25.4 mm/s)
  MoveL 309 to (266.15, 499.69, 1.82) mm, rotated rx -180 ry 0 rz 0 deg; joints [44.675, -46.774, 125.692, 45.33, -81.283, -7.585]
  MoveL 310 to (266.15, 499.69, -7.71) mm, rotated rx -180 ry 0 rz 0 deg; joints [44.681, -46.109, 125.559, 45.279, -81.657, -7.204]
  MoveC 311 to (266.34, 499.69, -8.16) mm, rotated rx 180 ry 0 rz 0 deg; joints [44.687, -46.081, 125.563, 45.282, -81.68, -7.182] to (266.79, 499.69, -8.35) mm, rotated rx -180 ry 0 rz 0 deg; joints [44.702, -46.077, 125.586, 45.294, -81.701, -7.164]
  Set speed (50.8 mm/s)
  MoveL 312 to (267.42, 499.69, -8.35) mm, rotated rx 180 ry 0 rz 0 deg; joints [44.723, -46.09, 125.622, 45.313, -81.72, -7.15]
  MoveC 313 to (267.87, 499.51, -8.35) mm, rotated rx -180 ry 0 rz 0 deg; joints [44.731, -46.102, 125.657, 45.319, -81.738, -7.135] to (268.06, 499.06, -8.35) mm, rotated rx 180 ry 0 rz 0 deg; joints [44.723, -46.114, 125.693, 45.308, -81.753, -7.117]
  MoveL 314 to (268.06, 473.66, -8.35) mm, rotated rx -180 ry 0 rz 0 deg; joints [43.87, -46.561, 127.087, 44.36, -82.321, -6.337]
  MoveL 315 to (217.26, 473.66, -8.35) mm, rotated rx 180 ry 0 rz 0 deg; joints [42.256, -45.537, 124.14, 42.938, -80.728, -7.465]
  MoveL 316 to (217.26, 524.46, -8.35) mm, rotated rx -180 ry 0 rz 0 deg; joints [43.933, -44.589, 121.351, 44.843, -79.649, -9.022]
  MoveL 317 to (268.06, 524.46, -8.35) mm, rotated rx -180 ry 0 rz 0 deg; joints [45.551, -45.644, 124.265, 46.24, -81.197, -7.921]
  MoveL 318 to (268.06, 499.06, -8.35) mm, rotated rx 180 ry 0 rz 0 deg; joints [44.723, -46.114, 125.693, 45.308, -81.753, -7.117]
  MoveC 319 to (267.87, 498.61, -8.35) mm, rotated rx -180 ry 0 rz 0 deg; joints [44.702, -46.118, 125.707, 45.286, -81.757, -7.107] to (267.42, 498.42, -8.35) mm, rotated rx 180 ry 0 rz 0 deg; joints [44.681, -46.113, 125.692, 45.266, -81.748, -7.111]
  MoveL 320 to (266.79, 498.42, -8.35) mm, rotated rx -180 ry 0 rz 0 deg; joints [44.66, -46.1, 125.656, 45.247, -81.729, -7.125]
  MoveC 321 to (266.34, 498.42, -8.16) mm, rotated rx 180 ry 0 rz 0 deg; joints [44.645, -46.104, 125.634, 45.235, -81.708, -7.142] to (266.15, 498.42, -7.72) mm, rotated rx 180 ry 0 rz 0 deg; joints [44.639, -46.132, 125.63, 45.232, -81.685, -7.164]
  Set speed (500.0 mm/s)
  MoveL 322 to (266.15, 498.42, 6) mm, rotated rx -180 ry 0 rz 0 deg; joints [44.63, -47.088, 125.819, 45.305, -81.144, -7.714]
  MoveL 323 to (393.15, 499.69, 6) mm, rotated rx 180 ry 0 rz 0 deg; joints [49.142, -49.399, 132.526, 49.422, -84.644, -4.943]
  Set speed (25.4 mm/s)
  MoveL 324 to (393.15, 499.69, -3.54) mm, rotated rx -180 ry 0 rz 0 deg; joints [49.149, -48.67, 132.388, 49.388, -85.029, -4.493]
  MoveC 325 to (393.34, 499.69, -3.99) mm, rotated rx 180 ry 0 rz 0 deg; joints [49.157, -48.639, 132.39, 49.394, -85.051, -4.468] to (393.79, 499.69, -4.17) mm, rotated rx 180 ry 0 rz 0 deg; joints [49.174, -48.632, 132.41, 49.409, -85.07, -4.449]
  Set speed (50.8 mm/s)
  MoveL 326 to (394.42, 499.69, -4.18) mm, rotated rx 180 ry 0 rz 0 deg; joints [49.198, -48.642, 132.442, 49.432, -85.086, -4.434]
  MoveC 327 to (394.87, 499.51, -4.17) mm, rotated rx 180 ry 0 rz 0 deg; joints [49.209, -48.652, 132.475, 49.441, -85.102, -4.417] to (395.06, 499.06, -4.18) mm, rotated rx 180 ry 0 rz 0 deg; joints [49.201, -48.662, 132.51, 49.432, -85.118, -4.398]
  MoveL 328 to (395.06, 473.66, -4.18) mm, rotated rx -180 ry 0 rz 0 deg; joints [48.355, -49.068, 133.957, 48.523, -85.738, -3.555]
  MoveL 329 to (344.26, 473.66, -4.17) mm, rotated rx -180 ry 0 rz 0 deg; joints [46.478, -48.249, 131.33, 46.76, -84.375, -4.763]
  MoveL 330 to (344.26, 524.46, -4.18) mm, rotated rx -180 ry 0 rz 0 deg; joints [48.154, -47.372, 128.449, 48.598, -83.196, -6.41]
  MoveL 331 to (395.06, 524.46, -4.18) mm, rotated rx -180 ry 0 rz 0 deg; joints [50.019, -48.231, 131.033, 50.322, -84.517, -5.262]
  MoveL 332 to (395.06, 499.06, -4.18) mm, rotated rx 180 ry 0 rz 0 deg; joints [49.201, -48.662, 132.51, 49.432, -85.118, -4.398]
  MoveC 333 to (394.87, 498.61, -4.18) mm, rotated rx -180 ry 0 rz 0 deg; joints [49.179, -48.667, 132.527, 49.409, -85.124, -4.387] to (394.42, 498.42, -4.18) mm, rotated rx -180 ry 0 rz 0 deg; joints [49.156, -48.663, 132.515, 49.387, -85.117, -4.391]
  MoveL 334 to (393.79, 498.42, -4.17) mm, rotated rx -180 ry 0 rz 0 deg; joints [49.132, -48.653, 132.483, 49.364, -85.101, -4.406]
  MoveC 335 to (393.34, 498.42, -3.99) mm, rotated rx -180 ry 0 rz 0 deg; joints [49.115, -48.66, 132.463, 49.348, -85.082, -4.425] to (393.15, 498.42, -3.54) mm, rotated rx -180 ry 0 rz 0 deg; joints [49.108, -48.691, 132.461, 49.343, -85.059, -4.451]
  Set speed (500.0 mm/s)
  MoveL 336 to (393.15, 498.42, 5) mm, rotated rx -180 ry 0 rz 0 deg; joints [49.102, -49.344, 132.585, 49.373, -84.714, -4.853]
  MoveL 337 to (393.15, 499.69, 5) mm, rotated rx -180 ry 0 rz 0 deg; joints [49.143, -49.322, 132.512, 49.418, -84.684, -4.896]
  Set speed (25.4 mm/s)
  MoveL 338 to (393.15, 499.69, 1.82) mm, rotated rx -180 ry 0 rz 0 deg; joints [49.145, -49.08, 132.466, 49.407, -84.813, -4.746]
  MoveL 339 to (393.15, 499.69, -7.72) mm, rotated rx 180 ry 0 rz 0 deg; joints [49.152, -48.351, 132.325, 49.375, -85.195, -4.299]
  MoveC 340 to (393.34, 499.69, -8.16) mm, rotated rx 180 ry 0 rz 0 deg; joints [49.16, -48.32, 132.327, 49.38, -85.218, -4.273] to (393.79, 499.69, -8.35) mm, rotated rx 180 ry 0 rz 0 deg; joints [49.177, -48.312, 132.347, 49.395, -85.237, -4.254]
  Set speed (50.8 mm/s)
  MoveL 341 to (394.42, 499.69, -8.35) mm, rotated rx -180 ry 0 rz 0 deg; joints [49.201, -48.322, 132.378, 49.418, -85.253, -4.239]
  MoveC 342 to (394.87, 499.51, -8.35) mm, rotated rx -180 ry 0 rz 0 deg; joints [49.212, -48.332, 132.411, 49.428, -85.269, -4.222] to (395.06, 499.06, -8.35) mm, rotated rx -180 ry 0 rz 0 deg; joints [49.204, -48.342, 132.447, 49.418, -85.285, -4.203]
  MoveL 343 to (395.06, 473.66, -8.35) mm, rotated rx 180 ry 0 rz 0 deg; joints [48.359, -48.741, 133.893, 48.512, -85.912, -3.358]
  MoveL 344 to (344.26, 473.66, -8.35) mm, rotated rx -180 ry 0 rz 0 deg; joints [46.481, -47.934, 131.267, 46.745, -84.548, -4.579]
  MoveL 345 to (344.26, 524.46, -8.35) mm, rotated rx -180 ry 0 rz 0 deg; joints [48.157, -47.07, 128.388, 48.58, -83.356, -6.228]
  MoveL 346 to (395.06, 524.46, -8.35) mm, rotated rx 180 ry 0 rz 0 deg; joints [50.022, -47.917, 130.97, 50.307, -84.677, -5.069]
  MoveL 347 to (395.06, 499.06, -8.35) mm, rotated rx -180 ry 0 rz 0 deg; joints [49.204, -48.342, 132.447, 49.418, -85.285, -4.203]
  MoveC 348 to (394.87, 498.61, -8.35) mm, rotated rx -180 ry 0 rz 0 deg; joints [49.183, -48.347, 132.463, 49.396, -85.291, -4.192] to (394.42, 498.42, -8.35) mm, rotated rx -180 ry 0 rz 0 deg; joints [49.159, -48.343, 132.451, 49.373, -85.284, -4.196]
  MoveL 349 to (393.79, 498.42, -8.35) mm, rotated rx 180 ry 0 rz 0 deg; joints [49.135, -48.333, 132.42, 49.351, -85.268, -4.211]
  MoveC 350 to (393.34, 498.42, -8.16) mm, rotated rx -180 ry 0 rz 0 deg; joints [49.118, -48.34, 132.4, 49.335, -85.249, -4.231] to (393.15, 498.42, -7.72) mm, rotated rx 180 ry 0 rz 0 deg; joints [49.111, -48.372, 132.398, 49.33, -85.226, -4.256]
  Set speed (500.0 mm/s)
  MoveL 351 to (393.15, 498.42, 6) mm, rotated rx -180 ry 0 rz 0 deg; joints [49.101, -49.421, 132.599, 49.377, -84.673, -4.901]
  MoveL 352 to (393.15, 313.35, 6) mm, rotated rx -180 ry 0 rz 0 deg; joints [42.222, -51.915, 142.447, 42.214, -89.524, 0.629]
  Set speed (25.4 mm/s)
  MoveL 353 to (393.15, 313.35, -3.54) mm, rotated rx 180 ry 0 rz 0 deg; joints [42.23, -51.058, 142.288, 42.219, -90.042, 1.099]
  MoveC 354 to (393.34, 313.36, -3.99) mm, rotated rx 180 ry 0 rz 0 deg; joints [42.237, -51.02, 142.29, 42.227, -90.071, 1.126] to (393.79, 313.35, -4.17) mm, rotated rx -180 ry 0 rz 0 deg; joints [42.254, -51.008, 142.311, 42.244, -90.095, 1.149]
  Set speed (50.8 mm/s)
  MoveL 355 to (394.42, 313.35, -4.17) mm, rotated rx -180 ry 0 rz 0 deg; joints [42.278, -51.015, 142.346, 42.268, -90.115, 1.167]
  MoveC 356 to (394.87, 313.17, -4.18) mm, rotated rx 180 ry 0 rz 0 deg; joints [42.288, -51.022, 142.379, 42.278, -90.134, 1.185] to (395.06, 312.72, -4.17) mm, rotated rx -180 ry 0 rz 0 deg; joints [42.276, -51.028, 142.41, 42.266, -90.153, 1.202]
  MoveL 357 to (395.06, 287.32, -4.17) mm, rotated rx 180 ry 0 rz 0 deg; joints [41.191, -51.238, 143.627, 41.188, -90.928, 1.846]
  MoveL 358 to (344.26, 287.32, -4.18) mm, rotated rx -180 ry 0 rz 0 deg; joints [39.333, -50.632, 140.808, 39.328, -89.266, 0.384]
  MoveL 359 to (344.26, 338.12, -4.17) mm, rotated rx 180 ry 0 rz 0 deg; joints [41.449, -50.114, 138.398, 41.474, -87.845, -0.864]
  MoveL 360 to (395.06, 338.12, -4.18) mm, rotated rx -180 ry 0 rz 0 deg; joints [43.324, -50.791, 141.161, 43.317, -89.399, 0.526]
  MoveL 361 to (395.06, 312.72, -4.17) mm, rotated rx -180 ry 0 rz 0 deg; joints [42.276, -51.028, 142.41, 42.266, -90.153, 1.202]
  MoveC 362 to (394.87, 312.27, -4.17) mm, rotated rx -180 ry 0 rz 0 deg; joints [42.25, -51.03, 142.422, 42.24, -90.161, 1.208] to (394.42, 312.09, -4.17) mm, rotated rx -180 ry 0 rz 0 deg; joints [42.225, -51.027, 142.407, 42.215, -90.153, 1.2]
  MoveL 363 to (393.79, 312.09, -4.18) mm, rotated rx 180 ry 0 rz 0 deg; joints [42.201, -51.019, 142.373, 42.191, -90.133, 1.182]
  MoveC 364 to (393.34, 312.08, -3.99) mm, rotated rx -180 ry 0 rz 0 deg; joints [42.184, -51.031, 142.352, 42.174, -90.11, 1.159] to (393.15, 312.08, -3.54) mm, rotated rx 180 ry 0 rz 0 deg; joints [42.176, -51.069, 142.35, 42.166, -90.08, 1.132]
  Set speed (500.0 mm/s)
  MoveL 365 to (393.15, 312.08, 5) mm, rotated rx -180 ry 0 rz 0 deg; joints [42.17, -51.838, 142.492, 42.161, -89.616, 0.712]
  MoveL 366 to (393.15, 313.36, 5) mm, rotated rx 180 ry 0 rz 0 deg; joints [42.223, -51.826, 142.43, 42.214, -89.578, 0.679]
  Set speed (25.4 mm/s)
  MoveL 367 to (393.15, 313.35, 1.82) mm, rotated rx 180 ry 0 rz 0 deg; joints [42.225, -51.54, 142.378, 42.216, -89.751, 0.836]
  MoveL 368 to (393.15, 313.35, -7.71) mm, rotated rx 180 ry 0 rz 0 deg; joints [42.233, -50.683, 142.216, 42.223, -90.266, 1.303]
  MoveC 369 to (393.34, 313.35, -8.16) mm, rotated rx -180 ry 0 rz 0 deg; joints [42.24, -50.644, 142.218, 42.231, -90.296, 1.33] to (393.79, 313.36, -8.35) mm, rotated rx -180 ry 0 rz 0 deg; joints [42.257, -50.633, 142.239, 42.248, -90.319, 1.352]
  Set speed (50.8 mm/s)
  MoveL 370 to (394.42, 313.35, -8.35) mm, rotated rx 180 ry 0 rz 0 deg; joints [42.282, -50.64, 142.273, 42.272, -90.339, 1.371]
  MoveC 371 to (394.87, 313.17, -8.35) mm, rotated rx -180 ry 0 rz 0 deg; joints [42.291, -50.646, 142.306, 42.282, -90.358, 1.389] to (395.06, 312.72, -8.35) mm, rotated rx -180 ry 0 rz 0 deg; joints [42.279, -50.652, 142.338, 42.27, -90.378, 1.406]
  MoveL 372 to (395.06, 287.32, -8.35) mm, rotated rx -180 ry 0 rz 0 deg; joints [41.195, -50.853, 143.553, 41.195, -91.162, 2.05]
  MoveL 373 to (344.26, 287.32, -8.35) mm, rotated rx -180 ry 0 rz 0 deg; joints [39.336, -50.267, 140.737, 39.329, -89.494, 0.57]
  MoveL 374 to (344.26, 338.12, -8.35) mm, rotated rx -180 ry 0 rz 0 deg; joints [41.452, -49.763, 138.33, 41.471, -88.056, -0.677]
  MoveL 375 to (395.06, 338.12, -8.35) mm, rotated rx -180 ry 0 rz 0 deg; joints [43.328, -50.423, 141.089, 43.319, -89.615, 0.729]
  MoveL 376 to (395.06, 312.72, -8.35) mm, rotated rx -180 ry 0 rz 0 deg; joints [42.279, -50.652, 142.338, 42.27, -90.378, 1.406]
  MoveC 377 to (394.87, 312.27, -8.35) mm, rotated rx -180 ry 0 rz 0 deg; joints [42.253, -50.654, 142.349, 42.244, -90.386, 1.412] to (394.42, 312.09, -8.35) mm, rotated rx -180 ry 0 rz 0 deg; joints [42.228, -50.651, 142.334, 42.219, -90.377, 1.404]
  MoveL 378 to (393.79, 312.09, -8.35) mm, rotated rx -180 ry 0 rz 0 deg; joints [42.204, -50.643, 142.3, 42.195, -90.358, 1.385]
  MoveC 379 to (393.34, 312.08, -8.16) mm, rotated rx -180 ry 0 rz 0 deg; joints [42.187, -50.655, 142.279, 42.178, -90.334, 1.363] to (393.15, 312.08, -7.72) mm, rotated rx -180 ry 0 rz 0 deg; joints [42.179, -50.693, 142.277, 42.17, -90.304, 1.336]
  Set speed (500.0 mm/s)
  MoveL 380 to (393.15, 312.08, 6) mm, rotated rx -180 ry 0 rz 0 deg; joints [42.169, -51.928, 142.508, 42.16, -89.561, 0.662]
  MoveL 381 to (266.15, 313.35, 6) mm, rotated rx 180 ry 0 rz 0 deg; joints [37.809, -49.982, 135.229, 37.945, -85.378, -2.649]
  Set speed (25.4 mm/s)
  MoveL 382 to (266.15, 313.35, -3.54) mm, rotated rx -180 ry 0 rz 0 deg; joints [37.816, -49.222, 135.085, 37.923, -85.864, -2.269]
  MoveC 383 to (266.34, 313.36, -3.99) mm, rotated rx -180 ry 0 rz 0 deg; joints [37.822, -49.19, 135.089, 37.927, -85.893, -2.247] to (266.79, 313.36, -4.17) mm, rotated rx -180 ry 0 rz 0 deg; joints [37.836, -49.183, 135.113, 37.94, -85.918, -2.229]
  Set speed (50.8 mm/s)
  MoveL 384 to (267.42, 313.36, -4.18) mm, rotated rx -180 ry 0 rz 0 deg; joints [37.857, -49.194, 135.151, 37.959, -85.94, -2.213]
  MoveC 385 to (267.87, 313.17, -4.17) mm, rotated rx -180 ry 0 rz 0 deg; joints [37.863, -49.203, 135.186, 37.965, -85.96, -2.198] to (268.06, 312.72, -4.17) mm, rotated rx -180 ry 0 rz 0 deg; joints [37.851, -49.212, 135.218, 37.951, -85.978, -2.183]
  MoveL 386 to (268.06, 287.32, -4.18) mm, rotated rx -180 ry 0 rz 0 deg; joints [36.798, -49.503, 136.367, 36.864, -86.62, -1.608]
  MoveL 387 to (217.26, 287.32, -4.17) mm, rotated rx 180 ry 0 rz 0 deg; joints [35.259, -48.61, 133.268, 35.42, -84.771, -2.821]
  MoveL 388 to (217.26, 338.12, -4.18) mm, rotated rx -180 ry 0 rz 0 deg; joints [37.303, -47.962, 130.98, 37.57, -83.584, -3.979]
  MoveL 389 to (268.06, 338.12, -4.18) mm, rotated rx 180 ry 0 rz 0 deg; joints [38.874, -48.899, 134.034, 39.018, -85.346, -2.789]
  MoveL 390 to (268.06, 312.72, -4.17) mm, rotated rx -180 ry 0 rz 0 deg; joints [37.851, -49.212, 135.218, 37.951, -85.978, -2.183]
  MoveC 391 to (267.87, 312.27, -4.17) mm, rotated rx -180 ry 0 rz 0 deg; joints [37.827, -49.214, 135.227, 37.927, -85.983, -2.177] to (267.42, 312.09, -4.18) mm, rotated rx -180 ry 0 rz 0 deg; joints [37.805, -49.209, 135.209, 37.906, -85.972, -2.184]
  MoveL 392 to (266.79, 312.09, -4.18) mm, rotated rx 180 ry 0 rz 0 deg; joints [37.785, -49.198, 135.171, 37.887, -85.95, -2.199]
  MoveC 393 to (266.34, 312.08, -3.99) mm, rotated rx -180 ry 0 rz 0 deg; joints [37.77, -49.205, 135.147, 37.874, -85.925, -2.218] to (266.15, 312.09, -3.54) mm, rotated rx 180 ry 0 rz 0 deg; joints [37.764, -49.238, 135.143, 37.869, -85.896, -2.24]
  Set speed (500.0 mm/s)
  MoveL 394 to (266.15, 312.09, 5) mm, rotated rx 180 ry 0 rz 0 deg; joints [37.758, -49.918, 135.272, 37.889, -85.46, -2.579]
  MoveL 395 to (266.15, 313.35, 5) mm, rotated rx 180 ry 0 rz 0 deg; joints [37.81, -49.902, 135.214, 37.943, -85.429, -2.609]
  Set speed (25.4 mm/s)
  MoveL 396 to (266.15, 313.35, 1.83) mm, rotated rx -180 ry 0 rz 0 deg; joints [37.812, -49.65, 135.167, 37.935, -85.591, -2.482]
  MoveL 397 to (266.15, 313.36, -7.72) mm, rotated rx 180 ry 0 rz 0 deg; joints [37.819, -48.89, 135.02, 37.914, -86.075, -2.105]
  MoveC 398 to (266.34, 313.36, -8.16) mm, rotated rx 180 ry 0 rz 0 deg; joints [37.825, -48.857, 135.023, 37.919, -86.104, -2.083] to (266.79, 313.35, -8.35) mm, rotated rx 180 ry 0 rz 0 deg; joints [37.839, -48.85, 135.047, 37.932, -86.129, -2.064]
  Set speed (50.8 mm/s)
  MoveL 399 to (267.42, 313.36, -8.35) mm, rotated rx -180 ry 0 rz 0 deg; joints [37.859, -48.861, 135.085, 37.951, -86.151, -2.049]
  MoveC 400 to (267.87, 313.17, -8.35) mm, rotated rx -180 ry 0 rz 0 deg; joints [37.866, -48.87, 135.12, 37.956, -86.171, -2.033] to (268.06, 312.72, -8.35) mm, rotated rx -180 ry 0 rz 0 deg; joints [37.854, -48.879, 135.152, 37.943, -86.189, -2.018]
  MoveL 401 to (268.06, 287.32, -8.35) mm, rotated rx -180 ry 0 rz 0 deg; joints [36.801, -49.163, 136.3, 36.857, -86.838, -1.445]
  MoveL 402 to (217.26, 287.32, -8.35) mm, rotated rx -180 ry 0 rz 0 deg; joints [35.262, -48.287, 133.203, 35.409, -84.982, -2.671]
  MoveL 403 to (217.26, 338.12, -8.35) mm, rotated rx 180 ry 0 rz 0 deg; joints [37.306, -47.649, 130.917, 37.556, -83.782, -3.826]
  MoveL 404 to (268.06, 338.12, -8.35) mm, rotated rx -180 ry 0 rz 0 deg; joints [38.877, -48.572, 133.969, 39.007, -85.55, -2.623]
  MoveL 405 to (268.06, 312.72, -8.35) mm, rotated rx -180 ry 0 rz 0 deg; joints [37.854, -48.879, 135.152, 37.943, -86.189, -2.018]
  MoveC 406 to (267.87, 312.27, -8.35) mm, rotated rx -180 ry 0 rz 0 deg; joints [37.829, -48.881, 135.161, 37.918, -86.194, -2.013] to (267.42, 312.08, -8.35) mm, rotated rx -180 ry 0 rz 0 deg; joints [37.807, -48.875, 135.143, 37.897, -86.183, -2.019]
  MoveL 407 to (266.79, 312.08, -8.35) mm, rotated rx 180 ry 0 rz 0 deg; joints [37.787, -48.865, 135.105, 37.878, -86.161, -2.035]
  MoveC 408 to (266.34, 312.08, -8.16) mm, rotated rx -180 ry 0 rz 0 deg; joints [37.773, -48.872, 135.082, 37.865, -86.136, -2.053] to (266.15, 312.08, -7.72) mm, rotated rx -180 ry 0 rz 0 deg; joints [37.767, -48.905, 135.078, 37.86, -86.107, -2.076]
  Set speed (500.0 mm/s)
  MoveL 409 to (266.15, 312.08, 6) mm, rotated rx -180 ry 0 rz 0 deg; joints [37.758, -49.998, 135.287, 37.891, -85.409, -2.619]
  MoveL 410 to (139.15, 313.35, 6) mm, rotated rx 180 ry 0 rz 0 deg; joints [34.127, -47.405, 127.304, 34.627, -80.786, -5.448]
  Set speed (25.4 mm/s)
  MoveL 411 to (139.15, 313.35, -3.54) mm, rotated rx 180 ry 0 rz 0 deg; joints [34.132, -46.727, 127.172, 34.584, -81.236, -5.135]
  MoveC 412 to (139.34, 313.36, -3.99) mm, rotated rx -180 ry 0 rz 0 deg; joints [34.138, -46.7, 127.177, 34.586, -81.264, -5.117] to (139.79, 313.36, -4.17) mm, rotated rx 180 ry 0 rz 0 deg; joints [34.15, -46.696, 127.204, 34.595, -81.29, -5.101]
  Set speed (50.8 mm/s)
  MoveL 413 to (140.42, 313.35, -4.17) mm, rotated rx 180 ry 0 rz 0 deg; joints [34.166, -46.71, 127.245, 34.61, -81.314, -5.088]
  MoveC 414 to (140.87, 313.17, -4.18) mm, rotated rx -180 ry 0 rz 0 deg; joints [34.171, -46.723, 127.283, 34.613, -81.335, -5.074] to (141.06, 312.72, -4.18) mm, rotated rx -180 ry 0 rz 0 deg; joints [34.158, -46.733, 127.314, 34.598, -81.351, -5.06]
  MoveL 415 to (141.06, 287.32, -4.17) mm, rotated rx -180 ry 0 rz 0 deg; joints [33.151, -47.075, 128.411, 33.522, -81.888, -4.5]
  MoveL 416 to (90.26, 287.32, -4.18) mm, rotated rx 180 ry 0 rz 0 deg; joints [31.866, -45.925, 125.033, 32.42, -79.9, -5.542]
  MoveL 417 to (90.26, 338.12, -4.17) mm, rotated rx 180 ry 0 rz 0 deg; joints [33.819, -45.192, 122.835, 34.546, -78.895, -6.698]
  MoveL 418 to (141.06, 338.12, -4.18) mm, rotated rx 180 ry 0 rz 0 deg; joints [35.142, -46.372, 126.181, 35.659, -80.816, -5.648]
  MoveL 419 to (141.06, 312.72, -4.18) mm, rotated rx -180 ry 0 rz 0 deg; joints [34.158, -46.733, 127.314, 34.598, -81.351, -5.06]
  MoveC 420 to (140.87, 312.27, -4.18) mm, rotated rx -180 ry 0 rz 0 deg; joints [34.136, -46.735, 127.322, 34.575, -81.354, -5.054] to (140.42, 312.09, -4.17) mm, rotated rx -180 ry 0 rz 0 deg; joints [34.117, -46.728, 127.301, 34.557, -81.341, -5.059]
  MoveL 421 to (139.79, 312.09, -4.18) mm, rotated rx -180 ry 0 rz 0 deg; joints [34.1, -46.714, 127.26, 34.542, -81.316, -5.072]
  MoveC 422 to (139.34, 312.08, -3.99) mm, rotated rx -180 ry 0 rz 0 deg; joints [34.088, -46.717, 127.233, 34.533, -81.291, -5.088] to (139.15, 312.08, -3.54) mm, rotated rx 180 ry 0 rz 0 deg; joints [34.083, -46.745, 127.227, 34.53, -81.263, -5.106]
  Set speed (500.0 mm/s)
  MoveL 423 to (139.15, 312.08, 5) mm, rotated rx -180 ry 0 rz 0 deg; joints [34.078, -47.352, 127.346, 34.569, -80.86, -5.386]
  MoveL 424 to (139.15, 313.35, 5) mm, rotated rx 180 ry 0 rz 0 deg; joints [34.127, -47.334, 127.29, 34.622, -80.834, -5.415]
  Set speed (25.4 mm/s)
  MoveL 425 to (139.15, 313.35, 1.82) mm, rotated rx -180 ry 0 rz 0 deg; joints [34.129, -47.109, 127.247, 34.608, -80.984, -5.31]
  MoveL 426 to (139.15, 313.36, -7.71) mm, rotated rx 180 ry 0 rz 0 deg; joints [34.135, -46.43, 127.111, 34.566, -81.431, -5]
  MoveC 427 to (139.34, 313.35, -8.16) mm, rotated rx -180 ry 0 rz 0 deg; joints [34.14, -46.402, 127.117, 34.568, -81.459, -4.981] to (139.79, 313.35, -8.35) mm, rotated rx -180 ry 0 rz 0 deg; joints [34.152, -46.399, 127.143, 34.578, -81.485, -4.966]
  Set speed (50.8 mm/s)
  MoveL 428 to (140.42, 313.36, -8.35) mm, rotated rx -180 ry 0 rz 0 deg; joints [34.169, -46.413, 127.184, 34.592, -81.509, -4.952]
  MoveC 429 to (140.87, 313.17, -8.35) mm, rotated rx -180 ry 0 rz 0 deg; joints [34.174, -46.425, 127.222, 34.595, -81.53, -4.938] to (141.06, 312.72, -8.35) mm, rotated rx 180 ry 0 rz 0 deg; joints [34.161, -46.435, 127.254, 34.58, -81.546, -4.924]
  MoveL 430 to (141.06, 287.32, -8.35) mm, rotated rx 180 ry 0 rz 0 deg; joints [33.154, -46.773, 128.35, 33.505, -82.089, -4.366]
  MoveL 431 to (90.26, 287.32, -8.35) mm, rotated rx -180 ry 0 rz 0 deg; joints [31.869, -45.636, 124.974, 32.401, -80.094, -5.418]
  MoveL 432 to (90.26, 338.12, -8.35) mm, rotated rx 180 ry 0 rz 0 deg; joints [33.821, -44.911, 122.777, 34.524, -79.079, -6.57]
  MoveL 433 to (141.06, 338.12, -8.35) mm, rotated rx 180 ry 0 rz 0 deg; joints [35.145, -46.079, 126.121, 35.639, -81.006, -5.511]
  MoveL 434 to (141.06, 312.72, -8.35) mm, rotated rx -180 ry 0 rz 0 deg; joints [34.161, -46.435, 127.254, 34.58, -81.546, -4.924]
  MoveC 435 to (140.87, 312.27, -8.35) mm, rotated rx -180 ry 0 rz 0 deg; joints [34.138, -46.437, 127.261, 34.557, -81.549, -4.918] to (140.42, 312.09, -8.35) mm, rotated rx 180 ry 0 rz 0 deg; joints [34.119, -46.43, 127.24, 34.539, -81.536, -4.924]
  MoveL 436 to (139.79, 312.08, -8.35) mm, rotated rx 180 ry 0 rz 0 deg; joints [34.102, -46.416, 127.199, 34.524, -81.512, -4.937]
  MoveC 437 to (139.34, 312.08, -8.16) mm, rotated rx -180 ry 0 rz 0 deg; joints [34.09, -46.42, 127.172, 34.515, -81.486, -4.953] to (139.15, 312.08, -7.72) mm, rotated rx -180 ry 0 rz 0 deg; joints [34.085, -46.448, 127.167, 34.512, -81.458, -4.971]
  Set speed (500.0 mm/s)
  MoveL 438 to (139.15, 312.08, 6) mm, rotated rx -180 ry 0 rz 0 deg; joints [34.077, -47.423, 127.36, 34.573, -80.813, -5.419]
  MoveL 439 to (139.15, 131.49, 6) mm, rotated rx -180 ry 0 rz 0 deg; joints [26.402, -49.528, 134.36, 26.526, -84.503, -2.033]
  Set speed (25.4 mm/s)
  MoveL 440 to (139.15, 131.49, -3.54) mm, rotated rx -180 ry 0 rz 0 deg; joints [26.407, -48.778, 134.217, 26.506, -85.046, -1.762]
  MoveC 441 to (139.34, 131.48, -3.99) mm, rotated rx -180 ry 0 rz 0 deg; joints [26.411, -48.747, 134.223, 26.509, -85.08, -1.746] to (139.79, 131.48, -4.17) mm, rotated rx 180 ry 0 rz 0 deg; joints [26.422, -48.741, 134.25, 26.518, -85.11, -1.731]
  Set speed (50.8 mm/s)
  MoveL 442 to (140.42, 131.49, -4.18) mm, rotated rx -180 ry 0 rz 0 deg; joints [26.436, -48.753, 134.293, 26.532, -85.138, -1.719]
  MoveC 443 to (140.87, 131.3, -4.17) mm, rotated rx -180 ry 0 rz 0 deg; joints [26.438, -48.764, 134.33, 26.532, -85.161, -1.707] to (141.06, 130.85, -4.17) mm, rotated rx -180 ry 0 rz 0 deg; joints [26.422, -48.771, 134.357, 26.515, -85.179, -1.697]
  MoveL 444 to (141.06, 105.45, -4.17) mm, rotated rx -180 ry 0 rz 0 deg; joints [25.244, -48.983, 135.187, 25.313, -85.697, -1.35]
  MoveL 445 to (90.26, 105.45, -4.18) mm, rotated rx -180 ry 0 rz 0 deg; joints [24.168, -47.955, 131.683, 24.331, -83.412, -2.308]
  MoveL 446 to (90.26, 156.25, -4.18) mm, rotated rx 180 ry 0 rz 0 deg; joints [26.429, -47.478, 130.022, 26.67, -82.459, -3.067]
  MoveL 447 to (141.06, 156.25, -4.17) mm, rotated rx 180 ry 0 rz 0 deg; joints [27.576, -48.542, 133.489, 27.699, -84.654, -2.074]
  MoveL 448 to (141.06, 130.85, -4.17) mm, rotated rx -180 ry 0 rz 0 deg; joints [26.422, -48.771, 134.357, 26.515, -85.179, -1.697]
  MoveC 449 to (140.87, 130.4, -4.17) mm, rotated rx -180 ry 0 rz 0 deg; joints [26.397, -48.771, 134.36, 26.49, -85.18, -1.694] to (140.42, 130.22, -4.18) mm, rotated rx -180 ry 0 rz 0 deg; joints [26.378, -48.764, 134.335, 26.472, -85.164, -1.7]
  MoveL 450 to (139.79, 130.22, -4.17) mm, rotated rx -180 ry 0 rz 0 deg; joints [26.363, -48.752, 134.293, 26.459, -85.136, -1.713]
  MoveC 451 to (139.34, 130.21, -3.99) mm, rotated rx 180 ry 0 rz 0 deg; joints [26.353, -48.758, 134.265, 26.45, -85.106, -1.727] to (139.15, 130.21, -3.54) mm, rotated rx 180 ry 0 rz 0 deg; joints [26.349, -48.789, 134.259, 26.447, -85.072, -1.744]
  Set speed (500.0 mm/s)
  MoveL 452 to (139.15, 130.22, 5) mm, rotated rx -180 ry 0 rz 0 deg; joints [26.344, -49.461, 134.388, 26.464, -84.586, -1.986]
  MoveL 453 to (139.15, 131.49, 5) mm, rotated rx 180 ry 0 rz 0 deg; joints [26.402, -49.449, 134.345, 26.523, -84.56, -2.005]
  Set speed (25.4 mm/s)
  MoveL 454 to (139.15, 131.49, 1.82) mm, rotated rx 180 ry 0 rz 0 deg; joints [26.404, -49.2, 134.298, 26.517, -84.742, -1.914]
  MoveL 455 to (139.15, 131.49, -7.72) mm, rotated rx -180 ry 0 rz 0 deg; joints [26.409, -48.45, 134.152, 26.499, -85.282, -1.644]
  MoveC 456 to (139.34, 131.48, -8.16) mm, rotated rx 180 ry 0 rz 0 deg; joints [26.414, -48.418, 134.157, 26.502, -85.315, -1.628] to (139.79, 131.49, -8.35) mm, rotated rx 180 ry 0 rz 0 deg; joints [26.424, -48.412, 134.185, 26.511, -85.345, -1.614]
  Set speed (50.8 mm/s)
  MoveL 457 to (140.42, 131.49, -8.35) mm, rotated rx -180 ry 0 rz 0 deg; joints [26.439, -48.424, 134.228, 26.524, -85.373, -1.601]
  MoveC 458 to (140.87, 131.3, -8.35) mm, rotated rx -180 ry 0 rz 0 deg; joints [26.44, -48.435, 134.264, 26.525, -85.397, -1.589] to (141.06, 130.85, -8.35) mm, rotated rx -180 ry 0 rz 0 deg; joints [26.424, -48.442, 134.292, 26.508, -85.415, -1.579]
  MoveL 459 to (141.06, 105.45, -8.35) mm, rotated rx 180 ry 0 rz 0 deg; joints [25.246, -48.65, 135.12, 25.307, -85.939, -1.236]
  MoveL 460 to (90.26, 105.45, -8.35) mm, rotated rx -180 ry 0 rz 0 deg; joints [24.17, -47.638, 131.62, 24.322, -83.642, -2.203]
  MoveL 461 to (90.26, 156.25, -8.35) mm, rotated rx -180 ry 0 rz 0 deg; joints [26.431, -47.169, 129.959, 26.658, -82.679, -2.956]
  MoveL 462 to (141.06, 156.25, -8.35) mm, rotated rx -180 ry 0 rz 0 deg; joints [27.578, -48.217, 133.424, 27.69, -84.884, -1.953]
  MoveL 463 to (141.06, 130.85, -8.35) mm, rotated rx 180 ry 0 rz 0 deg; joints [26.424, -48.442, 134.292, 26.508, -85.415, -1.579]
  MoveC 464 to (140.87, 130.4, -8.35) mm, rotated rx 180 ry 0 rz 0 deg; joints [26.399, -48.442, 134.294, 26.483, -85.416, -1.576] to (140.42, 130.21, -8.35) mm, rotated rx -180 ry 0 rz 0 deg; joints [26.38, -48.435, 134.27, 26.465, -85.4, -1.583]
  MoveL 465 to (139.79, 130.21, -8.35) mm, rotated rx 180 ry 0 rz 0 deg; joints [26.366, -48.423, 134.227, 26.451, -85.372, -1.596]
  MoveC 466 to (139.34, 130.22, -8.16) mm, rotated rx 180 ry 0 rz 0 deg; joints [26.356, -48.429, 134.2, 26.442, -85.341, -1.61] to (139.15, 130.22, -7.72) mm, rotated rx -180 ry 0 rz 0 deg; joints [26.351, -48.461, 134.194, 26.439, -85.308, -1.626]
  Set speed (500.0 mm/s)
  MoveL 467 to (139.15, 130.22, 6) mm, rotated rx -180 ry 0 rz 0 deg; joints [26.343, -49.539, 134.402, 26.466, -84.528, -2.015]
  MoveL 468 to (266.15, 131.48, 6) mm, rotated rx 180 ry 0 rz 0 deg; joints [29.613, -51.72, 142.68, 29.605, -89.964, 0.746]
  Set speed (25.4 mm/s)
  MoveL 469 to (266.15, 131.49, -3.54) mm, rotated rx -180 ry 0 rz 0 deg; joints [29.619, -50.859, 142.519, 29.613, -90.574, 1.093]
  MoveC 470 to (266.34, 131.48, -3.99) mm, rotated rx 180 ry 0 rz 0 deg; joints [29.625, -50.821, 142.523, 29.619, -90.611, 1.114] to (266.79, 131.49, -4.17) mm, rotated rx -180 ry 0 rz 0 deg; joints [29.637, -50.81, 142.548, 29.632, -90.642, 1.132]
  Set speed (50.8 mm/s)
  MoveL 471 to (267.42, 131.49, -4.18) mm, rotated rx -180 ry 0 rz 0 deg; joints [29.655, -50.818, 142.588, 29.65, -90.669, 1.148]
  MoveC 472 to (267.87, 131.3, -4.18) mm, rotated rx -180 ry 0 rz 0 deg; joints [29.659, -50.825, 142.623, 29.653, -90.694, 1.162] to (268.06, 130.85, -4.17) mm, rotated rx -180 ry 0 rz 0 deg; joints [29.642, -50.83, 142.651, 29.636, -90.713, 1.173]
  MoveL 473 to (268.06, 105.45, -4.17) mm, rotated rx -180 ry 0 rz 0 deg; joints [28.368, -50.974, 143.535, 28.37, -91.385, 1.489]
  MoveL 474 to (217.26, 105.45, -4.18) mm, rotated rx -180 ry 0 rz 0 deg; joints [27.037, -50.285, 140.265, 27.033, -89.113, 0.263]
  MoveL 475 to (217.26, 156.25, -4.17) mm, rotated rx -180 ry 0 rz 0 deg; joints [29.478, -49.915, 138.505, 29.492, -87.904, -0.422]
  MoveL 476 to (268.06, 156.25, -4.18) mm, rotated rx 180 ry 0 rz 0 deg; joints [30.884, -50.667, 141.728, 30.876, -90.041, 0.817]
  MoveL 477 to (268.06, 130.85, -4.17) mm, rotated rx -180 ry 0 rz 0 deg; joints [29.642, -50.83, 142.651, 29.636, -90.713, 1.173]
  MoveC 478 to (267.87, 130.4, -4.18) mm, rotated rx -180 ry 0 rz 0 deg; joints [29.614, -50.83, 142.655, 29.609, -90.717, 1.174] to (267.42, 130.21, -4.17) mm, rotated rx -180 ry 0 rz 0 deg; joints [29.592, -50.826, 142.634, 29.587, -90.703, 1.165]
  MoveL 479 to (266.79, 130.21, -4.18) mm, rotated rx -180 ry 0 rz 0 deg; joints [29.575, -50.817, 142.594, 29.569, -90.675, 1.149]
  MoveC 480 to (266.34, 130.22, -3.99) mm, rotated rx 180 ry 0 rz 0 deg; joints [29.562, -50.828, 142.569, 29.556, -90.644, 1.131] to (266.15, 130.21, -3.54) mm, rotated rx -180 ry 0 rz 0 deg; joints [29.556, -50.867, 142.565, 29.55, -90.608, 1.11]
  Set speed (500.0 mm/s)
  MoveL 481 to (266.15, 130.22, 5) mm, rotated rx -180 ry 0 rz 0 deg; joints [29.551, -51.639, 142.708, 29.543, -90.061, 0.8]
  MoveL 482 to (266.15, 131.49, 5) mm, rotated rx -180 ry 0 rz 0 deg; joints [29.614, -51.63, 142.663, 29.606, -90.029, 0.783]
  Set speed (25.4 mm/s)
  MoveL 483 to (266.15, 131.48, 1.83) mm, rotated rx -180 ry 0 rz 0 deg; joints [29.616, -51.343, 142.611, 29.608, -90.232, 0.898]
  MoveL 484 to (266.15, 131.49, -7.71) mm, rotated rx -180 ry 0 rz 0 deg; joints [29.622, -50.482, 142.446, 29.618, -90.838, 1.243]
  MoveC 485 to (266.34, 131.49, -8.16) mm, rotated rx 180 ry 0 rz 0 deg; joints [29.627, -50.444, 142.45, 29.623, -90.875, 1.264] to (266.79, 131.49, -8.35) mm, rotated rx -180 ry 0 rz 0 deg; joints [29.64, -50.433, 142.475, 29.636, -90.906, 1.282]
  Set speed (50.8 mm/s)
  MoveL 486 to (267.42, 131.49, -8.35) mm, rotated rx -180 ry 0 rz 0 deg; joints [29.658, -50.44, 142.515, 29.655, -90.933, 1.299]
  MoveC 487 to (267.87, 131.3, -8.35) mm, rotated rx -180 ry 0 rz 0 deg; joints [29.662, -50.447, 142.55, 29.658, -90.958, 1.313] to (268.06, 130.85, -8.35) mm, rotated rx -180 ry 0 rz 0 deg; joints [29.645, -50.452, 142.578, 29.641, -90.978, 1.324]
  MoveL 488 to (268.06, 105.45, -8.35) mm, rotated rx -180 ry 0 rz 0 deg; joints [28.371, -50.59, 143.461, 28.376, -91.657, 1.637]
  MoveL 489 to (217.26, 105.45, -8.35) mm, rotated rx 180 ry 0 rz 0 deg; joints [27.039, -49.923, 140.194, 27.034, -89.372, 0.396]
  MoveL 490 to (217.26, 156.25, -8.35) mm, rotated rx 180 ry 0 rz 0 deg; joints [29.48, -49.563, 138.436, 29.489, -88.149, -0.282]
  MoveL 491 to (268.06, 156.25, -8.35) mm, rotated rx -180 ry 0 rz 0 deg; joints [30.886, -50.295, 141.655, 30.879, -90.298, 0.97]
  MoveL 492 to (268.06, 130.85, -8.35) mm, rotated rx -180 ry 0 rz 0 deg; joints [29.645, -50.452, 142.578, 29.641, -90.978, 1.324]
  MoveC 493 to (267.87, 130.4, -8.35) mm, rotated rx 180 ry 0 rz 0 deg; joints [29.617, -50.452, 142.582, 29.614, -90.982, 1.325] to (267.42, 130.21, -8.35) mm, rotated rx 180 ry 0 rz 0 deg; joints [29.595, -50.448, 142.56, 29.592, -90.967, 1.315]
  MoveL 494 to (266.79, 130.21, -8.35) mm, rotated rx -180 ry 0 rz 0 deg; joints [29.577, -50.44, 142.52, 29.574, -90.94, 1.299]
  MoveC 495 to (266.34, 130.22, -8.16) mm, rotated rx -180 ry 0 rz 0 deg; joints [29.565, -50.451, 142.495, 29.561, -90.908, 1.281] to (266.15, 130.21, -7.72) mm, rotated rx -180 ry 0 rz 0 deg; joints [29.559, -50.489, 142.491, 29.555, -90.872, 1.26]
  Set speed (500.0 mm/s)
  MoveL 496 to (266.15, 130.22, 6) mm, rotated rx -180 ry 0 rz 0 deg; joints [29.55, -51.729, 142.725, 29.542, -89.997, 0.763]
  MoveL 497 to (393.15, 131.49, 6) mm, rotated rx -180 ry 0 rz 0 deg; joints [33.612, -52.987, 150.405, 33.767, -95.306, 4.388]
  Set speed (25.4 mm/s)
  MoveL 498 to (393.15, 131.49, -3.54) mm, rotated rx -180 ry 0 rz 0 deg; joints [33.619, -51.982, 150.221, 33.82, -95.987, 4.848]
  MoveC 499 to (393.34, 131.49, -3.99) mm, rotated rx 180 ry 0 rz 0 deg; joints [33.626, -51.935, 150.223, 33.83, -96.027, 4.876] to (393.79, 131.49, -4.18) mm, rotated rx 180 ry 0 rz 0 deg; joints [33.642, -51.917, 150.245, 33.848, -96.059, 4.9]
  Set speed (50.8 mm/s)
  MoveL 500 to (394.42, 131.48, -4.17) mm, rotated rx 180 ry 0 rz 0 deg; joints [33.665, -51.92, 150.282, 33.873, -96.086, 4.922]
  MoveC 501 to (394.87, 131.3, -4.18) mm, rotated rx -180 ry 0 rz 0 deg; joints [33.671, -51.922, 150.315, 33.881, -96.111, 4.94] to (395.06, 130.85, -4.18) mm, rotated rx 180 ry 0 rz 0 deg; joints [33.654, -51.923, 150.343, 33.865, -96.135, 4.953]
  MoveL 502 to (395.06, 105.45, -4.18) mm, rotated rx -180 ry 0 rz 0 deg; joints [32.283, -51.94, 151.298, 32.549, -97.035, 5.292]
  MoveL 503 to (344.26, 105.45, -4.17) mm, rotated rx -180 ry 0 rz 0 deg; joints [30.606, -51.697, 148.265, 30.716, -94.783, 3.623]
  MoveL 504 to (344.26, 156.25, -4.17) mm, rotated rx 180 ry 0 rz 0 deg; joints [33.233, -51.52, 146.377, 33.283, -93.193, 2.936]
  MoveL 505 to (395.06, 156.25, -4.17) mm, rotated rx -180 ry 0 rz 0 deg; joints [34.982, -51.882, 149.349, 35.142, -95.246, 4.563]
  MoveL 506 to (395.06, 130.85, -4.18) mm, rotated rx 180 ry 0 rz 0 deg; joints [33.654, -51.923, 150.343, 33.865, -96.135, 4.953]
  MoveC 507 to (394.87, 130.4, -4.18) mm, rotated rx -180 ry 0 rz 0 deg; joints [33.623, -51.923, 150.35, 33.835, -96.143, 4.953] to (394.42, 130.21, -4.17) mm, rotated rx -180 ry 0 rz 0 deg; joints [33.597, -51.922, 150.331, 33.808, -96.13, 4.94]
  MoveL 508 to (393.79, 130.22, -4.18) mm, rotated rx -180 ry 0 rz 0 deg; joints [33.575, -51.919, 150.294, 33.783, -96.104, 4.918]
  MoveC 509 to (393.34, 130.22, -3.99) mm, rotated rx -180 ry 0 rz 0 deg; joints [33.559, -51.937, 150.271, 33.765, -96.072, 4.894] to (393.15, 130.21, -3.54) mm, rotated rx 180 ry 0 rz 0 deg; joints [33.552, -51.983, 150.269, 33.755, -96.032, 4.866]
  Set speed (500.0 mm/s)
  MoveL 510 to (393.15, 130.22, 5) mm, rotated rx -180 ry 0 rz 0 deg; joints [33.545, -52.884, 150.435, 33.708, -95.421, 4.455]
  MoveL 511 to (393.15, 131.49, 5) mm, rotated rx 180 ry 0 rz 0 deg; joints [33.613, -52.881, 150.386, 33.773, -95.378, 4.437]
  Set speed (25.4 mm/s)
  MoveL 512 to (393.15, 131.48, 1.82) mm, rotated rx 180 ry 0 rz 0 deg; joints [33.615, -52.546, 150.326, 33.79, -95.606, 4.59]
  MoveL 513 to (393.15, 131.49, -7.72) mm, rotated rx -180 ry 0 rz 0 deg; joints [33.623, -51.543, 150.137, 33.845, -96.282, 5.047]
  MoveC 514 to (393.34, 131.48, -8.16) mm, rotated rx -180 ry 0 rz 0 deg; joints [33.63, -51.496, 150.138, 33.855, -96.321, 5.075] to (393.79, 131.48, -8.35) mm, rotated rx -180 ry 0 rz 0 deg; joints [33.646, -51.478, 150.161, 33.873, -96.353, 5.099]
  Set speed (50.8 mm/s)
  MoveL 515 to (394.42, 131.48, -8.35) mm, rotated rx -180 ry 0 rz 0 deg; joints [33.668, -51.481, 150.198, 33.898, -96.38, 5.121]
  MoveC 516 to (394.87, 131.3, -8.35) mm, rotated rx -180 ry 0 rz 0 deg; joints [33.674, -51.482, 150.231, 33.906, -96.406, 5.14] to (395.06, 130.85, -8.35) mm, rotated rx -180 ry 0 rz 0 deg; joints [33.657, -51.483, 150.259, 33.89, -96.429, 5.153]
  MoveL 517 to (395.06, 105.45, -8.35) mm, rotated rx -180 ry 0 rz 0 deg; joints [32.286, -51.491, 151.211, 32.577, -97.341, 5.489]
  MoveL 518 to (344.26, 105.45, -8.35) mm, rotated rx 180 ry 0 rz 0 deg; joints [30.609, -51.275, 148.184, 30.734, -95.075, 3.797]
  MoveL 519 to (344.26, 156.25, -8.35) mm, rotated rx 180 ry 0 rz 0 deg; joints [33.236, -51.114, 146.298, 33.296, -93.466, 3.116]
  MoveL 520 to (395.06, 156.25, -8.35) mm, rotated rx -180 ry 0 rz 0 deg; joints [34.985, -51.451, 149.266, 35.164, -95.53, 4.765]
  MoveL 521 to (395.06, 130.85, -8.35) mm, rotated rx -180 ry 0 rz 0 deg; joints [33.657, -51.483, 150.259, 33.89, -96.429, 5.153]
  MoveC 522 to (394.87, 130.4, -8.35) mm, rotated rx -180 ry 0 rz 0 deg; joints [33.626, -51.483, 150.265, 33.86, -96.438, 5.153] to (394.42, 130.21, -8.35) mm, rotated rx 180 ry 0 rz 0 deg; joints [33.601, -51.482, 150.246, 33.833, -96.425, 5.14]
  MoveL 523 to (393.79, 130.22, -8.35) mm, rotated rx 180 ry 0 rz 0 deg; joints [33.578, -51.479, 150.209, 33.808, -96.398, 5.117]
  MoveC 524 to (393.34, 130.21, -8.16) mm, rotated rx -180 ry 0 rz 0 deg; joints [33.562, -51.497, 150.187, 33.79, -96.366, 5.093] to (393.15, 130.21, -7.72) mm, rotated rx -180 ry 0 rz 0 deg; joints [33.555, -51.544, 150.185, 33.78, -96.327, 5.065]
  Set speed (500.0 mm/s)
  MoveL 525 to (393.15, 130.21, 6) mm, rotated rx 180 ry 0 rz 0 deg; joints [33.545, -52.989, 150.454, 33.702, -95.349, 4.407]
  MoveL 526 to (393.15, -54.85, 6) mm, rotated rx 180 ry 0 rz 0 deg; joints [22.587, -52.799, 156.44, 23.087, -101.711, 5.579]
  Set speed (25.4 mm/s)
  MoveL 527 to (393.15, -54.85, -3.54) mm, rotated rx 180 ry 0 rz 0 deg; joints [22.594, -51.642, 156.227, 23.174, -102.579, 5.96]
  MoveC 528 to (393.34, -54.85, -3.99) mm, rotated rx -180 ry 0 rz 0 deg; joints [22.599, -51.587, 156.228, 23.185, -102.63, 5.984] to (393.79, -54.85, -4.17) mm, rotated rx 180 ry 0 rz 0 deg; joints [22.611, -51.561, 156.252, 23.202, -102.675, 6.007]
  Set speed (50.8 mm/s)
  MoveL 529 to (394.42, -54.85, -4.18) mm, rotated rx -180 ry 0 rz 0 deg; joints [22.629, -51.556, 156.291, 23.223, -102.713, 6.029]
  MoveC 530 to (394.87, -55.04, -4.18) mm, rotated rx -180 ry 0 rz 0 deg; joints [22.629, -51.552, 156.324, 23.226, -102.747, 6.044] to (395.06, -55.49, -4.18) mm, rotated rx -180 ry 0 rz 0 deg; joints [22.604, -51.549, 156.347, 23.204, -102.774, 6.049]
  MoveL 531 to (395.06, -80.89, -4.18) mm, rotated rx -180 ry 0 rz 0 deg; joints [20.925, -51.43, 156.975, 21.554, -103.631, 5.923]
  MoveL 532 to (344.26, -80.89, -4.18) mm, rotated rx -180 ry 0 rz 0 deg; joints [19.698, -51.71, 153.745, 20.038, -100.454, 4.37]
  MoveL 533 to (344.26, -30.09, -4.18) mm, rotated rx 180 ry 0 rz 0 deg; joints [22.864, -51.785, 152.49, 23.158, -98.988, 4.462]
  MoveL 534 to (395.06, -30.09, -4.18) mm, rotated rx -180 ry 0 rz 0 deg; joints [24.244, -51.656, 155.672, 24.804, -101.893, 6.104]
  MoveL 535 to (395.06, -55.49, -4.18) mm, rotated rx -180 ry 0 rz 0 deg; joints [22.604, -51.549, 156.347, 23.204, -102.774, 6.049]
  MoveC 536 to (394.87, -55.94, -4.17) mm, rotated rx -180 ry 0 rz 0 deg; joints [22.57, -51.548, 156.347, 23.169, -102.778, 6.041] to (394.42, -56.12, -4.18) mm, rotated rx 180 ry 0 rz 0 deg; joints [22.546, -51.551, 156.324, 23.142, -102.757, 6.025]
  MoveL 537 to (393.79, -56.12, -4.17) mm, rotated rx 180 ry 0 rz 0 deg; joints [22.528, -51.555, 156.284, 23.12, -102.718, 6.003]
  MoveC 538 to (393.34, -56.12, -3.99) mm, rotated rx -180 ry 0 rz 0 deg; joints [22.516, -51.581, 156.261, 23.103, -102.674, 5.98] to (393.15, -56.12, -3.54) mm, rotated rx -180 ry 0 rz 0 deg; joints [22.511, -51.637, 156.259, 23.093, -102.622, 5.956]
  Set speed (500.0 mm/s)
  MoveL 539 to (393.15, -56.12, 5) mm, rotated rx 180 ry 0 rz 0 deg; joints [22.505, -52.673, 156.451, 23.015, -101.845, 5.616]
  MoveL 540 to (393.15, -54.85, 5) mm, rotated rx 180 ry 0 rz 0 deg; joints [22.587, -52.678, 156.418, 23.096, -101.803, 5.619]
  Set speed (25.4 mm/s)
  MoveL 541 to (393.15, -54.85, 1.82) mm, rotated rx -180 ry 0 rz 0 deg; joints [22.59, -52.292, 156.348, 23.125, -102.093, 5.746]
  MoveL 542 to (393.15, -54.85, -7.71) mm, rotated rx 180 ry 0 rz 0 deg; joints [22.597, -51.138, 156.13, 23.214, -102.952, 6.125]
  MoveC 543 to (393.34, -54.85, -8.16) mm, rotated rx -180 ry 0 rz 0 deg; joints [22.602, -51.083, 156.131, 23.224, -103.004, 6.149] to (393.79, -54.85, -8.35) mm, rotated rx -180 ry 0 rz 0 deg; joints [22.614, -51.057, 156.154, 23.241, -103.048, 6.172]
  Set speed (50.8 mm/s)
  MoveL 544 to (394.42, -54.85, -8.35) mm, rotated rx 180 ry 0 rz 0 deg; joints [22.632, -51.052, 156.194, 23.263, -103.087, 6.195]
  MoveC 545 to (394.87, -55.04, -8.35) mm, rotated rx -180 ry 0 rz 0 deg; joints [22.632, -51.047, 156.226, 23.266, -103.121, 6.21] to (395.06, -55.49, -8.35) mm, rotated rx 180 ry 0 rz 0 deg; joints [22.607, -51.043, 156.249, 23.244, -103.148, 6.215]
  MoveL 546 to (395.06, -80.89, -8.35) mm, rotated rx -180 ry 0 rz 0 deg; joints [20.927, -50.917, 156.875, 21.594, -104.015, 6.08]
  MoveL 547 to (344.26, -80.89, -8.35) mm, rotated rx -180 ry 0 rz 0 deg; joints [19.701, -51.235, 153.653, 20.066, -100.814, 4.504]
  MoveL 548 to (344.26, -30.09, -8.35) mm, rotated rx -180 ry 0 rz 0 deg; joints [22.867, -51.324, 152.401, 23.184, -99.33, 4.611]
  MoveL 549 to (395.06, -30.09, -8.35) mm, rotated rx -180 ry 0 rz 0 deg; joints [24.247, -51.159, 155.576, 24.843, -102.257, 6.277]
  MoveL 550 to (395.06, -55.49, -8.35) mm, rotated rx 180 ry 0 rz 0 deg; joints [22.607, -51.043, 156.249, 23.244, -103.148, 6.215]
  MoveC 551 to (394.87, -55.94, -8.35) mm, rotated rx 180 ry 0 rz 0 deg; joints [22.573, -51.043, 156.249, 23.209, -103.152, 6.206] to (394.42, -56.12, -8.35) mm, rotated rx 180 ry 0 rz 0 deg; joints [22.549, -51.046, 156.226, 23.182, -103.131, 6.19]
  MoveL 552 to (393.79, -56.12, -8.35) mm, rotated rx -180 ry 0 rz 0 deg; joints [22.531, -51.051, 156.187, 23.16, -103.092, 6.167]
  MoveC 553 to (393.34, -56.12, -8.16) mm, rotated rx -180 ry 0 rz 0 deg; joints [22.519, -51.077, 156.163, 23.143, -103.047, 6.144] to (393.15, -56.12, -7.72) mm, rotated rx -180 ry 0 rz 0 deg; joints [22.514, -51.132, 156.162, 23.132, -102.996, 6.12]
  Set speed (500.0 mm/s)
  MoveL 554 to (393.15, -56.12, 6) mm, rotated rx 180 ry 0 rz 0 deg; joints [22.504, -52.795, 156.473, 23.006, -101.753, 5.576]
  MoveL 555 to (266.15, -54.85, 6) mm, rotated rx 180 ry 0 rz 0 deg; joints [19.581, -52.507, 148.223, 19.638, -94.516, 2.191]
  Set speed (25.4 mm/s)
  MoveL 556 to (266.15, -54.85, -3.54) mm, rotated rx 180 ry 0 rz 0 deg; joints [19.587, -51.547, 148.046, 19.666, -95.252, 2.455]
  MoveC 557 to (266.34, -54.85, -3.99) mm, rotated rx -180 ry 0 rz 0 deg; joints [19.591, -51.504, 148.05, 19.672, -95.297, 2.472] to (266.79, -54.85, -4.17) mm, rotated rx -180 ry 0 rz 0 deg; joints [19.6, -51.488, 148.076, 19.682, -95.336, 2.487]
  Set speed (50.8 mm/s)
  MoveL 558 to (267.42, -54.85, -4.18) mm, rotated rx -180 ry 0 rz 0 deg; joints [19.613, -51.493, 148.118, 19.697, -95.371, 2.501]
  MoveC 559 to (267.87, -55.04, -4.18) mm, rotated rx -180 ry 0 rz 0 deg; joints [19.612, -51.496, 148.152, 19.696, -95.4, 2.511] to (268.06, -55.49, -4.17) mm, rotated rx -180 ry 0 rz 0 deg; joints [19.589, -51.498, 148.175, 19.675, -95.42, 2.516]
  MoveL 560 to (268.06, -80.89, -4.18) mm, rotated rx -180 ry 0 rz 0 deg; joints [18.098, -51.531, 148.747, 18.195, -95.989, 2.52]
  MoveL 561 to (217.26, -80.89, -4.17) mm, rotated rx -180 ry 0 rz 0 deg; joints [17.165, -51.095, 145.319, 17.186, -93.166, 1.519]
  MoveL 562 to (217.26, -30.09, -4.18) mm, rotated rx -180 ry 0 rz 0 deg; joints [19.991, -50.949, 144.168, 20, -92.156, 1.373]
  MoveL 563 to (268.06, -30.09, -4.18) mm, rotated rx -180 ry 0 rz 0 deg; joints [21.053, -51.454, 147.558, 21.125, -94.826, 2.469]
  MoveL 564 to (268.06, -55.49, -4.17) mm, rotated rx -180 ry 0 rz 0 deg; joints [19.589, -51.498, 148.175, 19.675, -95.42, 2.516]
  MoveC 565 to (267.87, -55.94, -4.18) mm, rotated rx -180 ry 0 rz 0 deg; joints [19.559, -51.498, 148.173, 19.644, -95.42, 2.512] to (267.42, -56.12, -4.17) mm, rotated rx -180 ry 0 rz 0 deg; joints [19.539, -51.495, 148.148, 19.624, -95.4, 2.503]
  MoveL 566 to (266.79, -56.12, -4.18) mm, rotated rx -180 ry 0 rz 0 deg; joints [19.526, -51.49, 148.106, 19.609, -95.365, 2.488]
  MoveC 567 to (266.34, -56.12, -3.99) mm, rotated rx 180 ry 0 rz 0 deg; joints [19.517, -51.506, 148.079, 19.599, -95.326, 2.473] to (266.15, -56.12, -3.54) mm, rotated rx -180 ry 0 rz 0 deg; joints [19.513, -51.549, 148.076, 19.593, -95.281, 2.457]
  Set speed (500.0 mm/s)
  MoveL 568 to (266.15, -56.12, 5) mm, rotated rx -180 ry 0 rz 0 deg; joints [19.508, -52.409, 148.235, 19.568, -94.622, 2.221]
  MoveL 569 to (266.15, -54.85, 5) mm, rotated rx -180 ry 0 rz 0 deg; joints [19.582, -52.406, 148.205, 19.641, -94.593, 2.219]
  Set speed (25.4 mm/s)
  MoveL 570 to (266.15, -54.85, 1.82) mm, rotated rx -180 ry 0 rz 0 deg; joints [19.583, -52.087, 148.147, 19.65, -94.839, 2.307]
  MoveL 571 to (266.15, -54.85, -7.72) mm, rotated rx -180 ry 0 rz 0 deg; joints [19.589, -51.128, 147.965, 19.679, -95.571, 2.57]
  MoveC 572 to (266.34, -54.85, -8.16) mm, rotated rx 180 ry 0 rz 0 deg; joints [19.593, -51.084, 147.969, 19.685, -95.615, 2.587] to (266.79, -54.85, -8.35) mm, rotated rx 180 ry 0 rz 0 deg; joints [19.603, -51.069, 147.995, 19.696, -95.654, 2.602]
  Set speed (50.8 mm/s)
  MoveL 573 to (267.42, -54.85, -8.35) mm, rotated rx -180 ry 0 rz 0 deg; joints [19.616, -51.073, 148.037, 19.71, -95.689, 2.616]
